//     PlcTask Inputs/GVL_iXlinker.EtherCAT_Master_ERxxxx.Beckhoff_ER6xxx.Beckhoff_ER6xxxEK1122.A_0005_ER6002_0002_0023.COM_TxPDO_Map_Inputs_Channel_2.Data_In[12] <-> COM TxPDO-Map Inputs Channel 2/Data In 12
//     PlcTask Inputs/GVL_iXlinker.EtherCAT_Master_ERxxxx.Beckhoff_ER6xxx.Beckhoff_ER6xxxEK1122.A_0005_ER6002_0002_0023.COM_TxPDO_Map_Inputs_Channel_2.Data_In[13] <-> COM TxPDO-Map Inputs Channel 2/Data In 13
//     PlcTask Inputs/GVL_iXlinker.EtherCAT_Master_ERxxxx.Beckhoff_ER6xxx.Beckhoff_ER6xxxEK1122.A_0005_ER6002_0002_0023.COM_TxPDO_Map_Inputs_Channel_2.Data_In[14] <-> COM TxPDO-Map Inputs Channel 2/Data In 14
//     PlcTask Inputs/GVL_iXlinker.EtherCAT_Master_ERxxxx.Beckhoff_ER6xxx.Beckhoff_ER6xxxEK1122.A_0005_ER6002_0002_0023.COM_TxPDO_Map_Inputs_Channel_2.Data_In[15] <-> COM TxPDO-Map Inputs Channel 2/Data In 15
//     PlcTask Inputs/GVL_iXlinker.EtherCAT_Master_ERxxxx.Beckhoff_ER6xxx.Beckhoff_ER6xxxEK1122.A_0005_ER6002_0002_0023.COM_TxPDO_Map_Inputs_Channel_2.Data_In[16] <-> COM TxPDO-Map Inputs Channel 2/Data In 16
//     PlcTask Inputs/GVL_iXlinker.EtherCAT_Master_ERxxxx.Beckhoff_ER6xxx.Beckhoff_ER6xxxEK1122.A_0005_ER6002_0002_0023.COM_TxPDO_Map_Inputs_Channel_2.Data_In[17] <-> COM TxPDO-Map Inputs Channel 2/Data In 17
//     PlcTask Inputs/GVL_iXlinker.EtherCAT_Master_ERxxxx.Beckhoff_ER6xxx.Beckhoff_ER6xxxEK1122.A_0005_ER6002_0002_0023.COM_TxPDO_Map_Inputs_Channel_2.Data_In[18] <-> COM TxPDO-Map Inputs Channel 2/Data In 18
//     PlcTask Inputs/GVL_iXlinker.EtherCAT_Master_ERxxxx.Beckhoff_ER6xxx.Beckhoff_ER6xxxEK1122.A_0005_ER6002_0002_0023.COM_TxPDO_Map_Inputs_Channel_2.Data_In[19] <-> COM TxPDO-Map Inputs Channel 2/Data In 19
//     PlcTask Inputs/GVL_iXlinker.EtherCAT_Master_ERxxxx.Beckhoff_ER6xxx.Beckhoff_ER6xxxEK1122.A_0005_ER6002_0002_0023.COM_TxPDO_Map_Inputs_Channel_2.Data_In[20] <-> COM TxPDO-Map Inputs Channel 2/Data In 20
//     PlcTask Inputs/GVL_iXlinker.EtherCAT_Master_ERxxxx.Beckhoff_ER6xxx.Beckhoff_ER6xxxEK1122.A_0005_ER6002_0002_0023.COM_TxPDO_Map_Inputs_Channel_2.Data_In[21] <-> COM TxPDO-Map Inputs Channel 2/Data In 21
//     PlcTask Outputs/GVL_iXlinker.EtherCAT_Master_ERxxxx.Beckhoff_ER6xxx.Beckhoff_ER6xxxEK1122.A_0005_ER6002_0002_0023.COM_RxPDO_Map_Outputs_Channel_1.Ctrl <-> COM RxPDO-Map Outputs Channel 1/Ctrl
//     PlcTask Outputs/GVL_iXlinker.EtherCAT_Master_ERxxxx.Beckhoff_ER6xxx.Beckhoff_ER6xxxEK1122.A_0005_ER6002_0002_0023.COM_RxPDO_Map_Outputs_Channel_2.Ctrl <-> COM RxPDO-Map Outputs Channel 2/Ctrl
//     PlcTask Outputs/GVL_iXlinker.EtherCAT_Master_ERxxxx.Beckhoff_ER6xxx.Beckhoff_ER6xxxEK1122.A_0005_ER6002_0002_0023.COM_RxPDO_Map_Outputs_Channel_1.Data_Out[0] <-> COM RxPDO-Map Outputs Channel 1/Data Out 0
//     PlcTask Outputs/GVL_iXlinker.EtherCAT_Master_ERxxxx.Beckhoff_ER6xxx.Beckhoff_ER6xxxEK1122.A_0005_ER6002_0002_0023.COM_RxPDO_Map_Outputs_Channel_1.Data_Out[1] <-> COM RxPDO-Map Outputs Channel 1/Data Out 1
//     PlcTask Outputs/GVL_iXlinker.EtherCAT_Master_ERxxxx.Beckhoff_ER6xxx.Beckhoff_ER6xxxEK1122.A_0005_ER6002_0002_0023.COM_RxPDO_Map_Outputs_Channel_1.Data_Out[2] <-> COM RxPDO-Map Outputs Channel 1/Data Out 2
//     PlcTask Outputs/GVL_iXlinker.EtherCAT_Master_ERxxxx.Beckhoff_ER6xxx.Beckhoff_ER6xxxEK1122.A_0005_ER6002_0002_0023.COM_RxPDO_Map_Outputs_Channel_1.Data_Out[3] <-> COM RxPDO-Map Outputs Channel 1/Data Out 3
//     PlcTask Outputs/GVL_iXlinker.EtherCAT_Master_ERxxxx.Beckhoff_ER6xxx.Beckhoff_ER6xxxEK1122.A_0005_ER6002_0002_0023.COM_RxPDO_Map_Outputs_Channel_1.Data_Out[4] <-> COM RxPDO-Map Outputs Channel 1/Data Out 4
//     PlcTask Outputs/GVL_iXlinker.EtherCAT_Master_ERxxxx.Beckhoff_ER6xxx.Beckhoff_ER6xxxEK1122.A_0005_ER6002_0002_0023.COM_RxPDO_Map_Outputs_Channel_1.Data_Out[5] <-> COM RxPDO-Map Outputs Channel 1/Data Out 5
//     PlcTask Outputs/GVL_iXlinker.EtherCAT_Master_ERxxxx.Beckhoff_ER6xxx.Beckhoff_ER6xxxEK1122.A_0005_ER6002_0002_0023.COM_RxPDO_Map_Outputs_Channel_1.Data_Out[6] <-> COM RxPDO-Map Outputs Channel 1/Data Out 6
//     PlcTask Outputs/GVL_iXlinker.EtherCAT_Master_ERxxxx.Beckhoff_ER6xxx.Beckhoff_ER6xxxEK1122.A_0005_ER6002_0002_0023.COM_RxPDO_Map_Outputs_Channel_1.Data_Out[7] <-> COM RxPDO-Map Outputs Channel 1/Data Out 7
//     PlcTask Outputs/GVL_iXlinker.EtherCAT_Master_ERxxxx.Beckhoff_ER6xxx.Beckhoff_ER6xxxEK1122.A_0005_ER6002_0002_0023.COM_RxPDO_Map_Outputs_Channel_1.Data_Out[8] <-> COM RxPDO-Map Outputs Channel 1/Data Out 8
//     PlcTask Outputs/GVL_iXlinker.EtherCAT_Master_ERxxxx.Beckhoff_ER6xxx.Beckhoff_ER6xxxEK1122.A_0005_ER6002_0002_0023.COM_RxPDO_Map_Outputs_Channel_1.Data_Out[9] <-> COM RxPDO-Map Outputs Channel 1/Data Out 9
//     PlcTask Outputs/GVL_iXlinker.EtherCAT_Master_ERxxxx.Beckhoff_ER6xxx.Beckhoff_ER6xxxEK1122.A_0005_ER6002_0002_0023.COM_RxPDO_Map_Outputs_Channel_1.Data_Out[10] <-> COM RxPDO-Map Outputs Channel 1/Data Out 10
//     PlcTask Outputs/GVL_iXlinker.EtherCAT_Master_ERxxxx.Beckhoff_ER6xxx.Beckhoff_ER6xxxEK1122.A_0005_ER6002_0002_0023.COM_RxPDO_Map_Outputs_Channel_1.Data_Out[11] <-> COM RxPDO-Map Outputs Channel 1/Data Out 11
//     PlcTask Outputs/GVL_iXlinker.EtherCAT_Master_ERxxxx.Beckhoff_ER6xxx.Beckhoff_ER6xxxEK1122.A_0005_ER6002_0002_0023.COM_RxPDO_Map_Outputs_Channel_1.Data_Out[12] <-> COM RxPDO-Map Outputs Channel 1/Data Out 12
//     PlcTask Outputs/GVL_iXlinker.EtherCAT_Master_ERxxxx.Beckhoff_ER6xxx.Beckhoff_ER6xxxEK1122.A_0005_ER6002_0002_0023.COM_RxPDO_Map_Outputs_Channel_1.Data_Out[13] <-> COM RxPDO-Map Outputs Channel 1/Data Out 13
//     PlcTask Outputs/GVL_iXlinker.EtherCAT_Master_ERxxxx.Beckhoff_ER6xxx.Beckhoff_ER6xxxEK1122.A_0005_ER6002_0002_0023.COM_RxPDO_Map_Outputs_Channel_1.Data_Out[14] <-> COM RxPDO-Map Outputs Channel 1/Data Out 14
//     PlcTask Outputs/GVL_iXlinker.EtherCAT_Master_ERxxxx.Beckhoff_ER6xxx.Beckhoff_ER6xxxEK1122.A_0005_ER6002_0002_0023.COM_RxPDO_Map_Outputs_Channel_1.Data_Out[15] <-> COM RxPDO-Map Outputs Channel 1/Data Out 15
//     PlcTask Outputs/GVL_iXlinker.EtherCAT_Master_ERxxxx.Beckhoff_ER6xxx.Beckhoff_ER6xxxEK1122.A_0005_ER6002_0002_0023.COM_RxPDO_Map_Outputs_Channel_1.Data_Out[16] <-> COM RxPDO-Map Outputs Channel 1/Data Out 16
//     PlcTask Outputs/GVL_iXlinker.EtherCAT_Master_ERxxxx.Beckhoff_ER6xxx.Beckhoff_ER6xxxEK1122.A_0005_ER6002_0002_0023.COM_RxPDO_Map_Outputs_Channel_1.Data_Out[17] <-> COM RxPDO-Map Outputs Channel 1/Data Out 17
//     PlcTask Outputs/GVL_iXlinker.EtherCAT_Master_ERxxxx.Beckhoff_ER6xxx.Beckhoff_ER6xxxEK1122.A_0005_ER6002_0002_0023.COM_RxPDO_Map_Outputs_Channel_1.Data_Out[18] <-> COM RxPDO-Map Outputs Channel 1/Data Out 18
//     PlcTask Outputs/GVL_iXlinker.EtherCAT_Master_ERxxxx.Beckhoff_ER6xxx.Beckhoff_ER6xxxEK1122.A_0005_ER6002_0002_0023.COM_RxPDO_Map_Outputs_Channel_1.Data_Out[19] <-> COM RxPDO-Map Outputs Channel 1/Data Out 19
//     PlcTask Outputs/GVL_iXlinker.EtherCAT_Master_ERxxxx.Beckhoff_ER6xxx.Beckhoff_ER6xxxEK1122.A_0005_ER6002_0002_0023.COM_RxPDO_Map_Outputs_Channel_1.Data_Out[20] <-> COM RxPDO-Map Outputs Channel 1/Data Out 20
//     PlcTask Outputs/GVL_iXlinker.EtherCAT_Master_ERxxxx.Beckhoff_ER6xxx.Beckhoff_ER6xxxEK1122.A_0005_ER6002_0002_0023.COM_RxPDO_Map_Outputs_Channel_1.Data_Out[21] <-> COM RxPDO-Map Outputs Channel 1/Data Out 21
//     PlcTask Outputs/GVL_iXlinker.EtherCAT_Master_ERxxxx.Beckhoff_ER6xxx.Beckhoff_ER6xxxEK1122.A_0005_ER6002_0002_0023.COM_RxPDO_Map_Outputs_Channel_2.Data_Out[0] <-> COM RxPDO-Map Outputs Channel 2/Data Out 0
//     PlcTask Outputs/GVL_iXlinker.EtherCAT_Master_ERxxxx.Beckhoff_ER6xxx.Beckhoff_ER6xxxEK1122.A_0005_ER6002_0002_0023.COM_RxPDO_Map_Outputs_Channel_2.Data_Out[1] <-> COM RxPDO-Map Outputs Channel 2/Data Out 1
//     PlcTask Outputs/GVL_iXlinker.EtherCAT_Master_ERxxxx.Beckhoff_ER6xxx.Beckhoff_ER6xxxEK1122.A_0005_ER6002_0002_0023.COM_RxPDO_Map_Outputs_Channel_2.Data_Out[2] <-> COM RxPDO-Map Outputs Channel 2/Data Out 2
//     PlcTask Outputs/GVL_iXlinker.EtherCAT_Master_ERxxxx.Beckhoff_ER6xxx.Beckhoff_ER6xxxEK1122.A_0005_ER6002_0002_0023.COM_RxPDO_Map_Outputs_Channel_2.Data_Out[3] <-> COM RxPDO-Map Outputs Channel 2/Data Out 3
//     PlcTask Outputs/GVL_iXlinker.EtherCAT_Master_ERxxxx.Beckhoff_ER6xxx.Beckhoff_ER6xxxEK1122.A_0005_ER6002_0002_0023.COM_RxPDO_Map_Outputs_Channel_2.Data_Out[4] <-> COM RxPDO-Map Outputs Channel 2/Data Out 4
//     PlcTask Outputs/GVL_iXlinker.EtherCAT_Master_ERxxxx.Beckhoff_ER6xxx.Beckhoff_ER6xxxEK1122.A_0005_ER6002_0002_0023.COM_RxPDO_Map_Outputs_Channel_2.Data_Out[5] <-> COM RxPDO-Map Outputs Channel 2/Data Out 5
//     PlcTask Outputs/GVL_iXlinker.EtherCAT_Master_ERxxxx.Beckhoff_ER6xxx.Beckhoff_ER6xxxEK1122.A_0005_ER6002_0002_0023.COM_RxPDO_Map_Outputs_Channel_2.Data_Out[6] <-> COM RxPDO-Map Outputs Channel 2/Data Out 6
//     PlcTask Outputs/GVL_iXlinker.EtherCAT_Master_ERxxxx.Beckhoff_ER6xxx.Beckhoff_ER6xxxEK1122.A_0005_ER6002_0002_0023.COM_RxPDO_Map_Outputs_Channel_2.Data_Out[7] <-> COM RxPDO-Map Outputs Channel 2/Data Out 7
//     PlcTask Outputs/GVL_iXlinker.EtherCAT_Master_ERxxxx.Beckhoff_ER6xxx.Beckhoff_ER6xxxEK1122.A_0005_ER6002_0002_0023.COM_RxPDO_Map_Outputs_Channel_2.Data_Out[8] <-> COM RxPDO-Map Outputs Channel 2/Data Out 8
//     PlcTask Outputs/GVL_iXlinker.EtherCAT_Master_ERxxxx.Beckhoff_ER6xxx.Beckhoff_ER6xxxEK1122.A_0005_ER6002_0002_0023.COM_RxPDO_Map_Outputs_Channel_2.Data_Out[9] <-> COM RxPDO-Map Outputs Channel 2/Data Out 9
//     PlcTask Outputs/GVL_iXlinker.EtherCAT_Master_ERxxxx.Beckhoff_ER6xxx.Beckhoff_ER6xxxEK1122.A_0005_ER6002_0002_0023.COM_RxPDO_Map_Outputs_Channel_2.Data_Out[10] <-> COM RxPDO-Map Outputs Channel 2/Data Out 10
//     PlcTask Outputs/GVL_iXlinker.EtherCAT_Master_ERxxxx.Beckhoff_ER6xxx.Beckhoff_ER6xxxEK1122.A_0005_ER6002_0002_0023.COM_RxPDO_Map_Outputs_Channel_2.Data_Out[11] <-> COM RxPDO-Map Outputs Channel 2/Data Out 11
//     PlcTask Outputs/GVL_iXlinker.EtherCAT_Master_ERxxxx.Beckhoff_ER6xxx.Beckhoff_ER6xxxEK1122.A_0005_ER6002_0002_0023.COM_RxPDO_Map_Outputs_Channel_2.Data_Out[12] <-> COM RxPDO-Map Outputs Channel 2/Data Out 12
//     PlcTask Outputs/GVL_iXlinker.EtherCAT_Master_ERxxxx.Beckhoff_ER6xxx.Beckhoff_ER6xxxEK1122.A_0005_ER6002_0002_0023.COM_RxPDO_Map_Outputs_Channel_2.Data_Out[13] <-> COM RxPDO-Map Outputs Channel 2/Data Out 13
//     PlcTask Outputs/GVL_iXlinker.EtherCAT_Master_ERxxxx.Beckhoff_ER6xxx.Beckhoff_ER6xxxEK1122.A_0005_ER6002_0002_0023.COM_RxPDO_Map_Outputs_Channel_2.Data_Out[14] <-> COM RxPDO-Map Outputs Channel 2/Data Out 14
//     PlcTask Outputs/GVL_iXlinker.EtherCAT_Master_ERxxxx.Beckhoff_ER6xxx.Beckhoff_ER6xxxEK1122.A_0005_ER6002_0002_0023.COM_RxPDO_Map_Outputs_Channel_2.Data_Out[15] <-> COM RxPDO-Map Outputs Channel 2/Data Out 15
//     PlcTask Outputs/GVL_iXlinker.EtherCAT_Master_ERxxxx.Beckhoff_ER6xxx.Beckhoff_ER6xxxEK1122.A_0005_ER6002_0002_0023.COM_RxPDO_Map_Outputs_Channel_2.Data_Out[16] <-> COM RxPDO-Map Outputs Channel 2/Data Out 16
//     PlcTask Outputs/GVL_iXlinker.EtherCAT_Master_ERxxxx.Beckhoff_ER6xxx.Beckhoff_ER6xxxEK1122.A_0005_ER6002_0002_0023.COM_RxPDO_Map_Outputs_Channel_2.Data_Out[17] <-> COM RxPDO-Map Outputs Channel 2/Data Out 17
//     PlcTask Outputs/GVL_iXlinker.EtherCAT_Master_ERxxxx.Beckhoff_ER6xxx.Beckhoff_ER6xxxEK1122.A_0005_ER6002_0002_0023.COM_RxPDO_Map_Outputs_Channel_2.Data_Out[18] <-> COM RxPDO-Map Outputs Channel 2/Data Out 18
//     PlcTask Outputs/GVL_iXlinker.EtherCAT_Master_ERxxxx.Beckhoff_ER6xxx.Beckhoff_ER6xxxEK1122.A_0005_ER6002_0002_0023.COM_RxPDO_Map_Outputs_Channel_2.Data_Out[19] <-> COM RxPDO-Map Outputs Channel 2/Data Out 19
//     PlcTask Outputs/GVL_iXlinker.EtherCAT_Master_ERxxxx.Beckhoff_ER6xxx.Beckhoff_ER6xxxEK1122.A_0005_ER6002_0002_0023.COM_RxPDO_Map_Outputs_Channel_2.Data_Out[20] <-> COM RxPDO-Map Outputs Channel 2/Data Out 20
//     PlcTask Outputs/GVL_iXlinker.EtherCAT_Master_ERxxxx.Beckhoff_ER6xxx.Beckhoff_ER6xxxEK1122.A_0005_ER6002_0002_0023.COM_RxPDO_Map_Outputs_Channel_2.Data_Out[21] <-> COM RxPDO-Map Outputs Channel 2/Data Out 21
//     PlcTask Inputs/GVL_iXlinker.EtherCAT_Master_ERxxxx.Beckhoff_ER6xxx.Beckhoff_ER6xxxEK1122.A_0005_ER6002_0002_0023.WcState.WcState <-> WcState/WcState
//     PlcTask Inputs/GVL_iXlinker.EtherCAT_Master_ERxxxx.Beckhoff_ER6xxx.Beckhoff_ER6xxxEK1122.A_0005_ER6002_0002_0023.WcState.InputToggle <-> WcState/InputToggle
//     PlcTask Inputs/GVL_iXlinker.EtherCAT_Master_ERxxxx.Beckhoff_ER6xxx.Beckhoff_ER6xxxEK1122.A_0005_ER6002_0002_0023.InfoData.AdsAddr <-> InfoData/AdsAddr
//     PlcTask Inputs/GVL_iXlinker.EtherCAT_Master_ERxxxx.Beckhoff_ER6xxx.Beckhoff_ER6xxxEK1122.A_0005_ER6002_0002_0023.InfoData.State <-> InfoData/State
//   PLC/PLC Instance <-> EtherCAT Master ERxxxx/Beckhoff ER7xxx
//     PlcTask Inputs/GVL_iXlinker.EtherCAT_Master_ERxxxx.Beckhoff_ER7xxx.InfoData.State <-> InfoData/State
//   PLC/PLC Instance <-> EtherCAT Master ERxxxx/Beckhoff ER7xxx/Beckhoff ER7xxxEK1122
//     PlcTask Inputs/GVL_iXlinker.EtherCAT_Master_ERxxxx.Beckhoff_ER7xxx.Beckhoff_ER7xxxEK1122.InfoData.State <-> InfoData/State
//   PLC/PLC Instance <-> EtherCAT Master ERxxxx/Beckhoff ER7xxx/Beckhoff ER7xxxEK1122/Beckhoff ER7xxxsub EK1100
//     PlcTask Inputs/GVL_iXlinker.EtherCAT_Master_ERxxxx.Beckhoff_ER7xxx.Beckhoff_ER7xxxEK1122.Beckhoff_ER7xxxsub_EK1100.InfoData.State <-> InfoData/State
//   PLC/PLC Instance <-> EtherCAT Master ERxxxx/Beckhoff ER7xxx/Beckhoff ER7xxxEK1122/A_0001(ER7041-0002-0024)
//     PlcTask Inputs/GVL_iXlinker.EtherCAT_Master_ERxxxx.Beckhoff_ER7xxx.Beckhoff_ER7xxxEK1122.A_0001_ER7041_0002_0024.ENC_Status_compact.Status/Latch_C_valid <-> ENC Status compact/Status/Latch C valid
//     PlcTask Inputs/GVL_iXlinker.EtherCAT_Master_ERxxxx.Beckhoff_ER7xxx.Beckhoff_ER7xxxEK1122.A_0001_ER7041_0002_0024.ENC_Status_compact.Status/Latch_extern_valid <-> ENC Status compact/Status/Latch extern valid
//     PlcTask Inputs/GVL_iXlinker.EtherCAT_Master_ERxxxx.Beckhoff_ER7xxx.Beckhoff_ER7xxxEK1122.A_0001_ER7041_0002_0024.ENC_Status_compact.Status/Set_counter_done <-> ENC Status compact/Status/Set counter done
//     PlcTask Inputs/GVL_iXlinker.EtherCAT_Master_ERxxxx.Beckhoff_ER7xxx.Beckhoff_ER7xxxEK1122.A_0001_ER7041_0002_0024.ENC_Status_compact.Status/Counter_underflow <-> ENC Status compact/Status/Counter underflow
//     PlcTask Inputs/GVL_iXlinker.EtherCAT_Master_ERxxxx.Beckhoff_ER7xxx.Beckhoff_ER7xxxEK1122.A_0001_ER7041_0002_0024.ENC_Status_compact.Status/Counter_overflow <-> ENC Status compact/Status/Counter overflow
//     PlcTask Inputs/GVL_iXlinker.EtherCAT_Master_ERxxxx.Beckhoff_ER7xxx.Beckhoff_ER7xxxEK1122.A_0001_ER7041_0002_0024.ENC_Status_compact.Status/Extrapolation_stall <-> ENC Status compact/Status/Extrapolation stall
//     PlcTask Inputs/GVL_iXlinker.EtherCAT_Master_ERxxxx.Beckhoff_ER7xxx.Beckhoff_ER7xxxEK1122.A_0001_ER7041_0002_0024.ENC_Status_compact.Status/Status_of_input_A <-> ENC Status compact/Status/Status of input A
//     PlcTask Inputs/GVL_iXlinker.EtherCAT_Master_ERxxxx.Beckhoff_ER7xxx.Beckhoff_ER7xxxEK1122.A_0001_ER7041_0002_0024.ENC_Status_compact.Status/Status_of_input_B <-> ENC Status compact/Status/Status of input B
//     PlcTask Inputs/GVL_iXlinker.EtherCAT_Master_ERxxxx.Beckhoff_ER7xxx.Beckhoff_ER7xxxEK1122.A_0001_ER7041_0002_0024.ENC_Status_compact.Status/Status_of_input_C <-> ENC Status compact/Status/Status of input C
//     PlcTask Inputs/GVL_iXlinker.EtherCAT_Master_ERxxxx.Beckhoff_ER7xxx.Beckhoff_ER7xxxEK1122.A_0001_ER7041_0002_0024.ENC_Status_compact.Status/Status_of_extern_latch <-> ENC Status compact/Status/Status of extern latch
//     PlcTask Inputs/GVL_iXlinker.EtherCAT_Master_ERxxxx.Beckhoff_ER7xxx.Beckhoff_ER7xxxEK1122.A_0001_ER7041_0002_0024.ENC_Status_compact.Status/Sync_error <-> ENC Status compact/Status/Sync error
//     PlcTask Inputs/GVL_iXlinker.EtherCAT_Master_ERxxxx.Beckhoff_ER7xxx.Beckhoff_ER7xxxEK1122.A_0001_ER7041_0002_0024.ENC_Status_compact.Status/TxPDO_Toggle <-> ENC Status compact/Status/TxPDO Toggle
//     PlcTask Inputs/GVL_iXlinker.EtherCAT_Master_ERxxxx.Beckhoff_ER7xxx.Beckhoff_ER7xxxEK1122.A_0001_ER7041_0002_0024.ENC_Status_compact.Counter_value <-> ENC Status compact/Counter value
//     PlcTask Inputs/GVL_iXlinker.EtherCAT_Master_ERxxxx.Beckhoff_ER7xxx.Beckhoff_ER7xxxEK1122.A_0001_ER7041_0002_0024.ENC_Status_compact.Latch_value <-> ENC Status compact/Latch value
//     PlcTask Inputs/GVL_iXlinker.EtherCAT_Master_ERxxxx.Beckhoff_ER7xxx.Beckhoff_ER7xxxEK1122.A_0001_ER7041_0002_0024.STM_Status.Status/Ready_to_enable <-> STM Status/Status/Ready to enable
//     PlcTask Inputs/GVL_iXlinker.EtherCAT_Master_ERxxxx.Beckhoff_ER7xxx.Beckhoff_ER7xxxEK1122.A_0001_ER7041_0002_0024.STM_Status.Status/Ready <-> STM Status/Status/Ready
//     PlcTask Inputs/GVL_iXlinker.EtherCAT_Master_ERxxxx.Beckhoff_ER7xxx.Beckhoff_ER7xxxEK1122.A_0001_ER7041_0002_0024.STM_Status.Status/Warning <-> STM Status/Status/Warning
//     PlcTask Inputs/GVL_iXlinker.EtherCAT_Master_ERxxxx.Beckhoff_ER7xxx.Beckhoff_ER7xxxEK1122.A_0001_ER7041_0002_0024.STM_Status.Status/Error <-> STM Status/Status/Error
//     PlcTask Inputs/GVL_iXlinker.EtherCAT_Master_ERxxxx.Beckhoff_ER7xxx.Beckhoff_ER7xxxEK1122.A_0001_ER7041_0002_0024.STM_Status.Status/Moving_positive <-> STM Status/Status/Moving positive
//     PlcTask Inputs/GVL_iXlinker.EtherCAT_Master_ERxxxx.Beckhoff_ER7xxx.Beckhoff_ER7xxxEK1122.A_0001_ER7041_0002_0024.STM_Status.Status/Moving_negative <-> STM Status/Status/Moving negative
//     PlcTask Inputs/GVL_iXlinker.EtherCAT_Master_ERxxxx.Beckhoff_ER7xxx.Beckhoff_ER7xxxEK1122.A_0001_ER7041_0002_0024.STM_Status.Status/Torque_reduced <-> STM Status/Status/Torque reduced
//     PlcTask Inputs/GVL_iXlinker.EtherCAT_Master_ERxxxx.Beckhoff_ER7xxx.Beckhoff_ER7xxxEK1122.A_0001_ER7041_0002_0024.STM_Status.Status/Digital_input_1 <-> STM Status/Status/Digital input 1
//     PlcTask Inputs/GVL_iXlinker.EtherCAT_Master_ERxxxx.Beckhoff_ER7xxx.Beckhoff_ER7xxxEK1122.A_0001_ER7041_0002_0024.STM_Status.Status/Digital_input_2 <-> STM Status/Status/Digital input 2
//     PlcTask Inputs/GVL_iXlinker.EtherCAT_Master_ERxxxx.Beckhoff_ER7xxx.Beckhoff_ER7xxxEK1122.A_0001_ER7041_0002_0024.STM_Status.Status/Sync_error <-> STM Status/Status/Sync error
//     PlcTask Inputs/GVL_iXlinker.EtherCAT_Master_ERxxxx.Beckhoff_ER7xxx.Beckhoff_ER7xxxEK1122.A_0001_ER7041_0002_0024.STM_Status.Status/TxPDO_Toggle <-> STM Status/Status/TxPDO Toggle
//     PlcTask Outputs/GVL_iXlinker.EtherCAT_Master_ERxxxx.Beckhoff_ER7xxx.Beckhoff_ER7xxxEK1122.A_0001_ER7041_0002_0024.ENC_Control_compact.Control/Enable_latch_C <-> ENC Control compact/Control/Enable latch C
//     PlcTask Outputs/GVL_iXlinker.EtherCAT_Master_ERxxxx.Beckhoff_ER7xxx.Beckhoff_ER7xxxEK1122.A_0001_ER7041_0002_0024.ENC_Control_compact.Control/Enable_latch_extern_on_positive_edge <-> ENC Control compact/Control/Enable latch extern on positive edge
//     PlcTask Outputs/GVL_iXlinker.EtherCAT_Master_ERxxxx.Beckhoff_ER7xxx.Beckhoff_ER7xxxEK1122.A_0001_ER7041_0002_0024.ENC_Control_compact.Control/Set_counter <-> ENC Control compact/Control/Set counter
//     PlcTask Outputs/GVL_iXlinker.EtherCAT_Master_ERxxxx.Beckhoff_ER7xxx.Beckhoff_ER7xxxEK1122.A_0001_ER7041_0002_0024.ENC_Control_compact.Control/Enable_latch_extern_on_negative_edge <-> ENC Control compact/Control/Enable latch extern on negative edge
//     PlcTask Outputs/GVL_iXlinker.EtherCAT_Master_ERxxxx.Beckhoff_ER7xxx.Beckhoff_ER7xxxEK1122.A_0001_ER7041_0002_0024.ENC_Control_compact.Set_counter_value <-> ENC Control compact/Set counter value
//     PlcTask Outputs/GVL_iXlinker.EtherCAT_Master_ERxxxx.Beckhoff_ER7xxx.Beckhoff_ER7xxxEK1122.A_0001_ER7041_0002_0024.STM_Control.Control/Enable <-> STM Control/Control/Enable
//     PlcTask Outputs/GVL_iXlinker.EtherCAT_Master_ERxxxx.Beckhoff_ER7xxx.Beckhoff_ER7xxxEK1122.A_0001_ER7041_0002_0024.STM_Control.Control/Reset <-> STM Control/Control/Reset
//     PlcTask Outputs/GVL_iXlinker.EtherCAT_Master_ERxxxx.Beckhoff_ER7xxx.Beckhoff_ER7xxxEK1122.A_0001_ER7041_0002_0024.STM_Control.Control/Reduce_torque <-> STM Control/Control/Reduce torque
//     PlcTask Outputs/GVL_iXlinker.EtherCAT_Master_ERxxxx.Beckhoff_ER7xxx.Beckhoff_ER7xxxEK1122.A_0001_ER7041_0002_0024.STM_Control.Control/Digital_output_1 <-> STM Control/Control/Digital output 1
//     PlcTask Outputs/GVL_iXlinker.EtherCAT_Master_ERxxxx.Beckhoff_ER7xxx.Beckhoff_ER7xxxEK1122.A_0001_ER7041_0002_0024.STM_Velocity.Velocity <-> STM Velocity/Velocity
//     PlcTask Inputs/GVL_iXlinker.EtherCAT_Master_ERxxxx.Beckhoff_ER7xxx.Beckhoff_ER7xxxEK1122.A_0001_ER7041_0002_0024.WcState.WcState <-> WcState/WcState
//     PlcTask Inputs/GVL_iXlinker.EtherCAT_Master_ERxxxx.Beckhoff_ER7xxx.Beckhoff_ER7xxxEK1122.A_0001_ER7041_0002_0024.WcState.InputToggle <-> WcState/InputToggle
//     PlcTask Inputs/GVL_iXlinker.EtherCAT_Master_ERxxxx.Beckhoff_ER7xxx.Beckhoff_ER7xxxEK1122.A_0001_ER7041_0002_0024.InfoData.AdsAddr <-> InfoData/AdsAddr
//     PlcTask Inputs/GVL_iXlinker.EtherCAT_Master_ERxxxx.Beckhoff_ER7xxx.Beckhoff_ER7xxxEK1122.A_0001_ER7041_0002_0024.InfoData.Chn0 <-> InfoData/Chn0
//     PlcTask Inputs/GVL_iXlinker.EtherCAT_Master_ERxxxx.Beckhoff_ER7xxx.Beckhoff_ER7xxxEK1122.A_0001_ER7041_0002_0024.InfoData.Chn1 <-> InfoData/Chn1
//     PlcTask Inputs/GVL_iXlinker.EtherCAT_Master_ERxxxx.Beckhoff_ER7xxx.Beckhoff_ER7xxxEK1122.A_0001_ER7041_0002_0024.InfoData.State <-> InfoData/State
//   PLC/PLC Instance <-> EtherCAT Master ERxxxx/Beckhoff ER7xxx/Beckhoff ER7xxxEK1122/A_0002(ER7041-0002-0025)
//     PlcTask Inputs/GVL_iXlinker.EtherCAT_Master_ERxxxx.Beckhoff_ER7xxx.Beckhoff_ER7xxxEK1122.A_0002_ER7041_0002_0025.ENC_Status_compact.Status/Latch_C_valid <-> ENC Status compact/Status/Latch C valid
//     PlcTask Inputs/GVL_iXlinker.EtherCAT_Master_ERxxxx.Beckhoff_ER7xxx.Beckhoff_ER7xxxEK1122.A_0002_ER7041_0002_0025.ENC_Status_compact.Status/Latch_extern_valid <-> ENC Status compact/Status/Latch extern valid
//     PlcTask Inputs/GVL_iXlinker.EtherCAT_Master_ERxxxx.Beckhoff_ER7xxx.Beckhoff_ER7xxxEK1122.A_0002_ER7041_0002_0025.ENC_Status_compact.Status/Set_counter_done <-> ENC Status compact/Status/Set counter done
//     PlcTask Inputs/GVL_iXlinker.EtherCAT_Master_ERxxxx.Beckhoff_ER7xxx.Beckhoff_ER7xxxEK1122.A_0002_ER7041_0002_0025.ENC_Status_compact.Status/Counter_underflow <-> ENC Status compact/Status/Counter underflow
//     PlcTask Inputs/GVL_iXlinker.EtherCAT_Master_ERxxxx.Beckhoff_ER7xxx.Beckhoff_ER7xxxEK1122.A_0002_ER7041_0002_0025.ENC_Status_compact.Status/Counter_overflow <-> ENC Status compact/Status/Counter overflow
//     PlcTask Inputs/GVL_iXlinker.EtherCAT_Master_ERxxxx.Beckhoff_ER7xxx.Beckhoff_ER7xxxEK1122.A_0002_ER7041_0002_0025.ENC_Status_compact.Status/Extrapolation_stall <-> ENC Status compact/Status/Extrapolation stall
//     PlcTask Inputs/GVL_iXlinker.EtherCAT_Master_ERxxxx.Beckhoff_ER7xxx.Beckhoff_ER7xxxEK1122.A_0002_ER7041_0002_0025.ENC_Status_compact.Status/Status_of_input_A <-> ENC Status compact/Status/Status of input A
//     PlcTask Inputs/GVL_iXlinker.EtherCAT_Master_ERxxxx.Beckhoff_ER7xxx.Beckhoff_ER7xxxEK1122.A_0002_ER7041_0002_0025.ENC_Status_compact.Status/Status_of_input_B <-> ENC Status compact/Status/Status of input B
//     PlcTask Inputs/GVL_iXlinker.EtherCAT_Master_ERxxxx.Beckhoff_ER7xxx.Beckhoff_ER7xxxEK1122.A_0002_ER7041_0002_0025.ENC_Status_compact.Status/Status_of_input_C <-> ENC Status compact/Status/Status of input C
//     PlcTask Inputs/GVL_iXlinker.EtherCAT_Master_ERxxxx.Beckhoff_ER7xxx.Beckhoff_ER7xxxEK1122.A_0002_ER7041_0002_0025.ENC_Status_compact.Status/Status_of_extern_latch <-> ENC Status compact/Status/Status of extern latch
//     PlcTask Inputs/GVL_iXlinker.EtherCAT_Master_ERxxxx.Beckhoff_ER7xxx.Beckhoff_ER7xxxEK1122.A_0002_ER7041_0002_0025.ENC_Status_compact.Status/Sync_error <-> ENC Status compact/Status/Sync error
//     PlcTask Inputs/GVL_iXlinker.EtherCAT_Master_ERxxxx.Beckhoff_ER7xxx.Beckhoff_ER7xxxEK1122.A_0002_ER7041_0002_0025.ENC_Status_compact.Status/TxPDO_Toggle <-> ENC Status compact/Status/TxPDO Toggle
//     PlcTask Inputs/GVL_iXlinker.EtherCAT_Master_ERxxxx.Beckhoff_ER7xxx.Beckhoff_ER7xxxEK1122.A_0002_ER7041_0002_0025.ENC_Status_compact.Counter_value <-> ENC Status compact/Counter value
//     PlcTask Inputs/GVL_iXlinker.EtherCAT_Master_ERxxxx.Beckhoff_ER7xxx.Beckhoff_ER7xxxEK1122.A_0002_ER7041_0002_0025.ENC_Status_compact.Latch_value <-> ENC Status compact/Latch value
//     PlcTask Inputs/GVL_iXlinker.EtherCAT_Master_ERxxxx.Beckhoff_ER7xxx.Beckhoff_ER7xxxEK1122.A_0002_ER7041_0002_0025.STM_Status.Status/Ready_to_enable <-> STM Status/Status/Ready to enable
//     PlcTask Inputs/GVL_iXlinker.EtherCAT_Master_ERxxxx.Beckhoff_ER7xxx.Beckhoff_ER7xxxEK1122.A_0002_ER7041_0002_0025.STM_Status.Status/Ready <-> STM Status/Status/Ready
//     PlcTask Inputs/GVL_iXlinker.EtherCAT_Master_ERxxxx.Beckhoff_ER7xxx.Beckhoff_ER7xxxEK1122.A_0002_ER7041_0002_0025.STM_Status.Status/Warning <-> STM Status/Status/Warning
//     PlcTask Inputs/GVL_iXlinker.EtherCAT_Master_ERxxxx.Beckhoff_ER7xxx.Beckhoff_ER7xxxEK1122.A_0002_ER7041_0002_0025.STM_Status.Status/Error <-> STM Status/Status/Error
//     PlcTask Inputs/GVL_iXlinker.EtherCAT_Master_ERxxxx.Beckhoff_ER7xxx.Beckhoff_ER7xxxEK1122.A_0002_ER7041_0002_0025.STM_Status.Status/Moving_positive <-> STM Status/Status/Moving positive
//     PlcTask Inputs/GVL_iXlinker.EtherCAT_Master_ERxxxx.Beckhoff_ER7xxx.Beckhoff_ER7xxxEK1122.A_0002_ER7041_0002_0025.STM_Status.Status/Moving_negative <-> STM Status/Status/Moving negative
//     PlcTask Inputs/GVL_iXlinker.EtherCAT_Master_ERxxxx.Beckhoff_ER7xxx.Beckhoff_ER7xxxEK1122.A_0002_ER7041_0002_0025.STM_Status.Status/Torque_reduced <-> STM Status/Status/Torque reduced
//     PlcTask Inputs/GVL_iXlinker.EtherCAT_Master_ERxxxx.Beckhoff_ER7xxx.Beckhoff_ER7xxxEK1122.A_0002_ER7041_0002_0025.STM_Status.Status/Digital_input_1 <-> STM Status/Status/Digital input 1
//     PlcTask Inputs/GVL_iXlinker.EtherCAT_Master_ERxxxx.Beckhoff_ER7xxx.Beckhoff_ER7xxxEK1122.A_0002_ER7041_0002_0025.STM_Status.Status/Digital_input_2 <-> STM Status/Status/Digital input 2
//     PlcTask Inputs/GVL_iXlinker.EtherCAT_Master_ERxxxx.Beckhoff_ER7xxx.Beckhoff_ER7xxxEK1122.A_0002_ER7041_0002_0025.STM_Status.Status/Sync_error <-> STM Status/Status/Sync error
//     PlcTask Inputs/GVL_iXlinker.EtherCAT_Master_ERxxxx.Beckhoff_ER7xxx.Beckhoff_ER7xxxEK1122.A_0002_ER7041_0002_0025.STM_Status.Status/TxPDO_Toggle <-> STM Status/Status/TxPDO Toggle
//     PlcTask Outputs/GVL_iXlinker.EtherCAT_Master_ERxxxx.Beckhoff_ER7xxx.Beckhoff_ER7xxxEK1122.A_0002_ER7041_0002_0025.ENC_Control_compact.Control/Enable_latch_C <-> ENC Control compact/Control/Enable latch C
//     PlcTask Outputs/GVL_iXlinker.EtherCAT_Master_ERxxxx.Beckhoff_ER7xxx.Beckhoff_ER7xxxEK1122.A_0002_ER7041_0002_0025.ENC_Control_compact.Control/Enable_latch_extern_on_positive_edge <-> ENC Control compact/Control/Enable latch extern on positive edge
//     PlcTask Outputs/GVL_iXlinker.EtherCAT_Master_ERxxxx.Beckhoff_ER7xxx.Beckhoff_ER7xxxEK1122.A_0002_ER7041_0002_0025.ENC_Control_compact.Control/Set_counter <-> ENC Control compact/Control/Set counter
//     PlcTask Outputs/GVL_iXlinker.EtherCAT_Master_ERxxxx.Beckhoff_ER7xxx.Beckhoff_ER7xxxEK1122.A_0002_ER7041_0002_0025.ENC_Control_compact.Control/Enable_latch_extern_on_negative_edge <-> ENC Control compact/Control/Enable latch extern on negative edge
//     PlcTask Outputs/GVL_iXlinker.EtherCAT_Master_ERxxxx.Beckhoff_ER7xxx.Beckhoff_ER7xxxEK1122.A_0002_ER7041_0002_0025.ENC_Control_compact.Set_counter_value <-> ENC Control compact/Set counter value
//     PlcTask Outputs/GVL_iXlinker.EtherCAT_Master_ERxxxx.Beckhoff_ER7xxx.Beckhoff_ER7xxxEK1122.A_0002_ER7041_0002_0025.STM_Control.Control/Enable <-> STM Control/Control/Enable
//     PlcTask Outputs/GVL_iXlinker.EtherCAT_Master_ERxxxx.Beckhoff_ER7xxx.Beckhoff_ER7xxxEK1122.A_0002_ER7041_0002_0025.STM_Control.Control/Reset <-> STM Control/Control/Reset
//     PlcTask Outputs/GVL_iXlinker.EtherCAT_Master_ERxxxx.Beckhoff_ER7xxx.Beckhoff_ER7xxxEK1122.A_0002_ER7041_0002_0025.STM_Control.Control/Reduce_torque <-> STM Control/Control/Reduce torque
//     PlcTask Outputs/GVL_iXlinker.EtherCAT_Master_ERxxxx.Beckhoff_ER7xxx.Beckhoff_ER7xxxEK1122.A_0002_ER7041_0002_0025.STM_Control.Control/Digital_output_1 <-> STM Control/Control/Digital output 1
//     PlcTask Outputs/GVL_iXlinker.EtherCAT_Master_ERxxxx.Beckhoff_ER7xxx.Beckhoff_ER7xxxEK1122.A_0002_ER7041_0002_0025.STM_Velocity.Velocity <-> STM Velocity/Velocity
//     PlcTask Inputs/GVL_iXlinker.EtherCAT_Master_ERxxxx.Beckhoff_ER7xxx.Beckhoff_ER7xxxEK1122.A_0002_ER7041_0002_0025.WcState.WcState <-> WcState/WcState
//     PlcTask Inputs/GVL_iXlinker.EtherCAT_Master_ERxxxx.Beckhoff_ER7xxx.Beckhoff_ER7xxxEK1122.A_0002_ER7041_0002_0025.WcState.InputToggle <-> WcState/InputToggle
//     PlcTask Inputs/GVL_iXlinker.EtherCAT_Master_ERxxxx.Beckhoff_ER7xxx.Beckhoff_ER7xxxEK1122.A_0002_ER7041_0002_0025.InfoData.AdsAddr <-> InfoData/AdsAddr
//     PlcTask Inputs/GVL_iXlinker.EtherCAT_Master_ERxxxx.Beckhoff_ER7xxx.Beckhoff_ER7xxxEK1122.A_0002_ER7041_0002_0025.InfoData.Chn0 <-> InfoData/Chn0
//     PlcTask Inputs/GVL_iXlinker.EtherCAT_Master_ERxxxx.Beckhoff_ER7xxx.Beckhoff_ER7xxxEK1122.A_0002_ER7041_0002_0025.InfoData.Chn1 <-> InfoData/Chn1
//     PlcTask Inputs/GVL_iXlinker.EtherCAT_Master_ERxxxx.Beckhoff_ER7xxx.Beckhoff_ER7xxxEK1122.A_0002_ER7041_0002_0025.InfoData.State <-> InfoData/State
//   PLC/PLC Instance <-> EtherCAT Master ERxxxx/Beckhoff ER7xxx/Beckhoff ER7xxxEK1122/A_0003(ER7041-1002-0024)
//     PlcTask Inputs/GVL_iXlinker.EtherCAT_Master_ERxxxx.Beckhoff_ER7xxx.Beckhoff_ER7xxxEK1122.A_0003_ER7041_1002_0024.ENC_Status_compact.Status/Latch_C_valid <-> ENC Status compact/Status/Latch C valid
//     PlcTask Inputs/GVL_iXlinker.EtherCAT_Master_ERxxxx.Beckhoff_ER7xxx.Beckhoff_ER7xxxEK1122.A_0003_ER7041_1002_0024.ENC_Status_compact.Status/Latch_extern_valid <-> ENC Status compact/Status/Latch extern valid
//     PlcTask Inputs/GVL_iXlinker.EtherCAT_Master_ERxxxx.Beckhoff_ER7xxx.Beckhoff_ER7xxxEK1122.A_0003_ER7041_1002_0024.ENC_Status_compact.Status/Set_counter_done <-> ENC Status compact/Status/Set counter done
//     PlcTask Inputs/GVL_iXlinker.EtherCAT_Master_ERxxxx.Beckhoff_ER7xxx.Beckhoff_ER7xxxEK1122.A_0003_ER7041_1002_0024.ENC_Status_compact.Status/Counter_underflow <-> ENC Status compact/Status/Counter underflow
//     PlcTask Inputs/GVL_iXlinker.EtherCAT_Master_ERxxxx.Beckhoff_ER7xxx.Beckhoff_ER7xxxEK1122.A_0003_ER7041_1002_0024.ENC_Status_compact.Status/Counter_overflow <-> ENC Status compact/Status/Counter overflow
//     PlcTask Inputs/GVL_iXlinker.EtherCAT_Master_ERxxxx.Beckhoff_ER7xxx.Beckhoff_ER7xxxEK1122.A_0003_ER7041_1002_0024.ENC_Status_compact.Status/Extrapolation_stall <-> ENC Status compact/Status/Extrapolation stall
//     PlcTask Inputs/GVL_iXlinker.EtherCAT_Master_ERxxxx.Beckhoff_ER7xxx.Beckhoff_ER7xxxEK1122.A_0003_ER7041_1002_0024.ENC_Status_compact.Status/Status_of_input_A <-> ENC Status compact/Status/Status of input A
//     PlcTask Inputs/GVL_iXlinker.EtherCAT_Master_ERxxxx.Beckhoff_ER7xxx.Beckhoff_ER7xxxEK1122.A_0003_ER7041_1002_0024.ENC_Status_compact.Status/Status_of_input_B <-> ENC Status compact/Status/Status of input B
//     PlcTask Inputs/GVL_iXlinker.EtherCAT_Master_ERxxxx.Beckhoff_ER7xxx.Beckhoff_ER7xxxEK1122.A_0003_ER7041_1002_0024.ENC_Status_compact.Status/Status_of_input_C <-> ENC Status compact/Status/Status of input C
//     PlcTask Inputs/GVL_iXlinker.EtherCAT_Master_ERxxxx.Beckhoff_ER7xxx.Beckhoff_ER7xxxEK1122.A_0003_ER7041_1002_0024.ENC_Status_compact.Status/Status_of_extern_latch <-> ENC Status compact/Status/Status of extern latch
//     PlcTask Inputs/GVL_iXlinker.EtherCAT_Master_ERxxxx.Beckhoff_ER7xxx.Beckhoff_ER7xxxEK1122.A_0003_ER7041_1002_0024.ENC_Status_compact.Status/Sync_error <-> ENC Status compact/Status/Sync error
//     PlcTask Inputs/GVL_iXlinker.EtherCAT_Master_ERxxxx.Beckhoff_ER7xxx.Beckhoff_ER7xxxEK1122.A_0003_ER7041_1002_0024.ENC_Status_compact.Status/TxPDO_Toggle <-> ENC Status compact/Status/TxPDO Toggle
//     PlcTask Inputs/GVL_iXlinker.EtherCAT_Master_ERxxxx.Beckhoff_ER7xxx.Beckhoff_ER7xxxEK1122.A_0003_ER7041_1002_0024.ENC_Status_compact.Counter_value <-> ENC Status compact/Counter value
//     PlcTask Inputs/GVL_iXlinker.EtherCAT_Master_ERxxxx.Beckhoff_ER7xxx.Beckhoff_ER7xxxEK1122.A_0003_ER7041_1002_0024.ENC_Status_compact.Latch_value <-> ENC Status compact/Latch value
//     PlcTask Inputs/GVL_iXlinker.EtherCAT_Master_ERxxxx.Beckhoff_ER7xxx.Beckhoff_ER7xxxEK1122.A_0003_ER7041_1002_0024.STM_Status.Status/Ready_to_enable <-> STM Status/Status/Ready to enable
//     PlcTask Inputs/GVL_iXlinker.EtherCAT_Master_ERxxxx.Beckhoff_ER7xxx.Beckhoff_ER7xxxEK1122.A_0003_ER7041_1002_0024.STM_Status.Status/Ready <-> STM Status/Status/Ready
//     PlcTask Inputs/GVL_iXlinker.EtherCAT_Master_ERxxxx.Beckhoff_ER7xxx.Beckhoff_ER7xxxEK1122.A_0003_ER7041_1002_0024.STM_Status.Status/Warning <-> STM Status/Status/Warning
//     PlcTask Inputs/GVL_iXlinker.EtherCAT_Master_ERxxxx.Beckhoff_ER7xxx.Beckhoff_ER7xxxEK1122.A_0003_ER7041_1002_0024.STM_Status.Status/Error <-> STM Status/Status/Error
//     PlcTask Inputs/GVL_iXlinker.EtherCAT_Master_ERxxxx.Beckhoff_ER7xxx.Beckhoff_ER7xxxEK1122.A_0003_ER7041_1002_0024.STM_Status.Status/Moving_positive <-> STM Status/Status/Moving positive
//     PlcTask Inputs/GVL_iXlinker.EtherCAT_Master_ERxxxx.Beckhoff_ER7xxx.Beckhoff_ER7xxxEK1122.A_0003_ER7041_1002_0024.STM_Status.Status/Moving_negative <-> STM Status/Status/Moving negative
//     PlcTask Inputs/GVL_iXlinker.EtherCAT_Master_ERxxxx.Beckhoff_ER7xxx.Beckhoff_ER7xxxEK1122.A_0003_ER7041_1002_0024.STM_Status.Status/Torque_reduced <-> STM Status/Status/Torque reduced
//     PlcTask Inputs/GVL_iXlinker.EtherCAT_Master_ERxxxx.Beckhoff_ER7xxx.Beckhoff_ER7xxxEK1122.A_0003_ER7041_1002_0024.STM_Status.Status/Digital_input_1 <-> STM Status/Status/Digital input 1
//     PlcTask Inputs/GVL_iXlinker.EtherCAT_Master_ERxxxx.Beckhoff_ER7xxx.Beckhoff_ER7xxxEK1122.A_0003_ER7041_1002_0024.STM_Status.Status/Digital_input_2 <-> STM Status/Status/Digital input 2
//     PlcTask Inputs/GVL_iXlinker.EtherCAT_Master_ERxxxx.Beckhoff_ER7xxx.Beckhoff_ER7xxxEK1122.A_0003_ER7041_1002_0024.STM_Status.Status/Sync_error <-> STM Status/Status/Sync error
//     PlcTask Inputs/GVL_iXlinker.EtherCAT_Master_ERxxxx.Beckhoff_ER7xxx.Beckhoff_ER7xxxEK1122.A_0003_ER7041_1002_0024.STM_Status.Status/TxPDO_Toggle <-> STM Status/Status/TxPDO Toggle
//     PlcTask Outputs/GVL_iXlinker.EtherCAT_Master_ERxxxx.Beckhoff_ER7xxx.Beckhoff_ER7xxxEK1122.A_0003_ER7041_1002_0024.ENC_Control_compact.Control/Enable_latch_C <-> ENC Control compact/Control/Enable latch C
//     PlcTask Outputs/GVL_iXlinker.EtherCAT_Master_ERxxxx.Beckhoff_ER7xxx.Beckhoff_ER7xxxEK1122.A_0003_ER7041_1002_0024.ENC_Control_compact.Control/Enable_latch_extern_on_positive_edge <-> ENC Control compact/Control/Enable latch extern on positive edge
//     PlcTask Outputs/GVL_iXlinker.EtherCAT_Master_ERxxxx.Beckhoff_ER7xxx.Beckhoff_ER7xxxEK1122.A_0003_ER7041_1002_0024.ENC_Control_compact.Control/Set_counter <-> ENC Control compact/Control/Set counter
//     PlcTask Outputs/GVL_iXlinker.EtherCAT_Master_ERxxxx.Beckhoff_ER7xxx.Beckhoff_ER7xxxEK1122.A_0003_ER7041_1002_0024.ENC_Control_compact.Control/Enable_latch_extern_on_negative_edge <-> ENC Control compact/Control/Enable latch extern on negative edge
//     PlcTask Outputs/GVL_iXlinker.EtherCAT_Master_ERxxxx.Beckhoff_ER7xxx.Beckhoff_ER7xxxEK1122.A_0003_ER7041_1002_0024.ENC_Control_compact.Set_counter_value <-> ENC Control compact/Set counter value
//     PlcTask Outputs/GVL_iXlinker.EtherCAT_Master_ERxxxx.Beckhoff_ER7xxx.Beckhoff_ER7xxxEK1122.A_0003_ER7041_1002_0024.STM_Control.Control/Enable <-> STM Control/Control/Enable
//     PlcTask Outputs/GVL_iXlinker.EtherCAT_Master_ERxxxx.Beckhoff_ER7xxx.Beckhoff_ER7xxxEK1122.A_0003_ER7041_1002_0024.STM_Control.Control/Reset <-> STM Control/Control/Reset
//     PlcTask Outputs/GVL_iXlinker.EtherCAT_Master_ERxxxx.Beckhoff_ER7xxx.Beckhoff_ER7xxxEK1122.A_0003_ER7041_1002_0024.STM_Control.Control/Reduce_torque <-> STM Control/Control/Reduce torque
//     PlcTask Outputs/GVL_iXlinker.EtherCAT_Master_ERxxxx.Beckhoff_ER7xxx.Beckhoff_ER7xxxEK1122.A_0003_ER7041_1002_0024.STM_Control.Control/Digital_output_1 <-> STM Control/Control/Digital output 1
//     PlcTask Outputs/GVL_iXlinker.EtherCAT_Master_ERxxxx.Beckhoff_ER7xxx.Beckhoff_ER7xxxEK1122.A_0003_ER7041_1002_0024.STM_Velocity.Velocity <-> STM Velocity/Velocity
//     PlcTask Inputs/GVL_iXlinker.EtherCAT_Master_ERxxxx.Beckhoff_ER7xxx.Beckhoff_ER7xxxEK1122.A_0003_ER7041_1002_0024.WcState.WcState <-> WcState/WcState
//     PlcTask Inputs/GVL_iXlinker.EtherCAT_Master_ERxxxx.Beckhoff_ER7xxx.Beckhoff_ER7xxxEK1122.A_0003_ER7041_1002_0024.WcState.InputToggle <-> WcState/InputToggle
//     PlcTask Inputs/GVL_iXlinker.EtherCAT_Master_ERxxxx.Beckhoff_ER7xxx.Beckhoff_ER7xxxEK1122.A_0003_ER7041_1002_0024.InfoData.AdsAddr <-> InfoData/AdsAddr
//     PlcTask Inputs/GVL_iXlinker.EtherCAT_Master_ERxxxx.Beckhoff_ER7xxx.Beckhoff_ER7xxxEK1122.A_0003_ER7041_1002_0024.InfoData.Chn0 <-> InfoData/Chn0
//     PlcTask Inputs/GVL_iXlinker.EtherCAT_Master_ERxxxx.Beckhoff_ER7xxx.Beckhoff_ER7xxxEK1122.A_0003_ER7041_1002_0024.InfoData.Chn1 <-> InfoData/Chn1
//     PlcTask Inputs/GVL_iXlinker.EtherCAT_Master_ERxxxx.Beckhoff_ER7xxx.Beckhoff_ER7xxxEK1122.A_0003_ER7041_1002_0024.InfoData.State <-> InfoData/State
//   PLC/PLC Instance <-> EtherCAT Master ERxxxx/Beckhoff ER7xxx/Beckhoff ER7xxxEK1122/A_0004(ER7041-1002-0025)
//     PlcTask Inputs/GVL_iXlinker.EtherCAT_Master_ERxxxx.Beckhoff_ER7xxx.Beckhoff_ER7xxxEK1122.A_0004_ER7041_1002_0025.ENC_Status_compact.Status/Latch_C_valid <-> ENC Status compact/Status/Latch C valid
//     PlcTask Inputs/GVL_iXlinker.EtherCAT_Master_ERxxxx.Beckhoff_ER7xxx.Beckhoff_ER7xxxEK1122.A_0004_ER7041_1002_0025.ENC_Status_compact.Status/Latch_extern_valid <-> ENC Status compact/Status/Latch extern valid
//     PlcTask Inputs/GVL_iXlinker.EtherCAT_Master_ERxxxx.Beckhoff_ER7xxx.Beckhoff_ER7xxxEK1122.A_0004_ER7041_1002_0025.ENC_Status_compact.Status/Set_counter_done <-> ENC Status compact/Status/Set counter done
//     PlcTask Inputs/GVL_iXlinker.EtherCAT_Master_ERxxxx.Beckhoff_ER7xxx.Beckhoff_ER7xxxEK1122.A_0004_ER7041_1002_0025.ENC_Status_compact.Status/Counter_underflow <-> ENC Status compact/Status/Counter underflow
//     PlcTask Inputs/GVL_iXlinker.EtherCAT_Master_ERxxxx.Beckhoff_ER7xxx.Beckhoff_ER7xxxEK1122.A_0004_ER7041_1002_0025.ENC_Status_compact.Status/Counter_overflow <-> ENC Status compact/Status/Counter overflow
//     PlcTask Inputs/GVL_iXlinker.EtherCAT_Master_ERxxxx.Beckhoff_ER7xxx.Beckhoff_ER7xxxEK1122.A_0004_ER7041_1002_0025.ENC_Status_compact.Status/Extrapolation_stall <-> ENC Status compact/Status/Extrapolation stall
//     PlcTask Inputs/GVL_iXlinker.EtherCAT_Master_ERxxxx.Beckhoff_ER7xxx.Beckhoff_ER7xxxEK1122.A_0004_ER7041_1002_0025.ENC_Status_compact.Status/Status_of_input_A <-> ENC Status compact/Status/Status of input A
//     PlcTask Inputs/GVL_iXlinker.EtherCAT_Master_ERxxxx.Beckhoff_ER7xxx.Beckhoff_ER7xxxEK1122.A_0004_ER7041_1002_0025.ENC_Status_compact.Status/Status_of_input_B <-> ENC Status compact/Status/Status of input B
//     PlcTask Inputs/GVL_iXlinker.EtherCAT_Master_ERxxxx.Beckhoff_ER7xxx.Beckhoff_ER7xxxEK1122.A_0004_ER7041_1002_0025.ENC_Status_compact.Status/Status_of_input_C <-> ENC Status compact/Status/Status of input C
//     PlcTask Inputs/GVL_iXlinker.EtherCAT_Master_ERxxxx.Beckhoff_ER7xxx.Beckhoff_ER7xxxEK1122.A_0004_ER7041_1002_0025.ENC_Status_compact.Status/Status_of_extern_latch <-> ENC Status compact/Status/Status of extern latch
//     PlcTask Inputs/GVL_iXlinker.EtherCAT_Master_ERxxxx.Beckhoff_ER7xxx.Beckhoff_ER7xxxEK1122.A_0004_ER7041_1002_0025.ENC_Status_compact.Status/Sync_error <-> ENC Status compact/Status/Sync error
//     PlcTask Inputs/GVL_iXlinker.EtherCAT_Master_ERxxxx.Beckhoff_ER7xxx.Beckhoff_ER7xxxEK1122.A_0004_ER7041_1002_0025.ENC_Status_compact.Status/TxPDO_Toggle <-> ENC Status compact/Status/TxPDO Toggle
//     PlcTask Inputs/GVL_iXlinker.EtherCAT_Master_ERxxxx.Beckhoff_ER7xxx.Beckhoff_ER7xxxEK1122.A_0004_ER7041_1002_0025.ENC_Status_compact.Counter_value <-> ENC Status compact/Counter value
//     PlcTask Inputs/GVL_iXlinker.EtherCAT_Master_ERxxxx.Beckhoff_ER7xxx.Beckhoff_ER7xxxEK1122.A_0004_ER7041_1002_0025.ENC_Status_compact.Latch_value <-> ENC Status compact/Latch value
//     PlcTask Inputs/GVL_iXlinker.EtherCAT_Master_ERxxxx.Beckhoff_ER7xxx.Beckhoff_ER7xxxEK1122.A_0004_ER7041_1002_0025.STM_Status.Status/Ready_to_enable <-> STM Status/Status/Ready to enable
//     PlcTask Inputs/GVL_iXlinker.EtherCAT_Master_ERxxxx.Beckhoff_ER7xxx.Beckhoff_ER7xxxEK1122.A_0004_ER7041_1002_0025.STM_Status.Status/Ready <-> STM Status/Status/Ready
//     PlcTask Inputs/GVL_iXlinker.EtherCAT_Master_ERxxxx.Beckhoff_ER7xxx.Beckhoff_ER7xxxEK1122.A_0004_ER7041_1002_0025.STM_Status.Status/Warning <-> STM Status/Status/Warning
//     PlcTask Inputs/GVL_iXlinker.EtherCAT_Master_ERxxxx.Beckhoff_ER7xxx.Beckhoff_ER7xxxEK1122.A_0004_ER7041_1002_0025.STM_Status.Status/Error <-> STM Status/Status/Error
//     PlcTask Inputs/GVL_iXlinker.EtherCAT_Master_ERxxxx.Beckhoff_ER7xxx.Beckhoff_ER7xxxEK1122.A_0004_ER7041_1002_0025.STM_Status.Status/Moving_positive <-> STM Status/Status/Moving positive
//     PlcTask Inputs/GVL_iXlinker.EtherCAT_Master_ERxxxx.Beckhoff_ER7xxx.Beckhoff_ER7xxxEK1122.A_0004_ER7041_1002_0025.STM_Status.Status/Moving_negative <-> STM Status/Status/Moving negative
//     PlcTask Inputs/GVL_iXlinker.EtherCAT_Master_ERxxxx.Beckhoff_ER7xxx.Beckhoff_ER7xxxEK1122.A_0004_ER7041_1002_0025.STM_Status.Status/Torque_reduced <-> STM Status/Status/Torque reduced
//     PlcTask Inputs/GVL_iXlinker.EtherCAT_Master_ERxxxx.Beckhoff_ER7xxx.Beckhoff_ER7xxxEK1122.A_0004_ER7041_1002_0025.STM_Status.Status/Digital_input_1 <-> STM Status/Status/Digital input 1
//     PlcTask Inputs/GVL_iXlinker.EtherCAT_Master_ERxxxx.Beckhoff_ER7xxx.Beckhoff_ER7xxxEK1122.A_0004_ER7041_1002_0025.STM_Status.Status/Digital_input_2 <-> STM Status/Status/Digital input 2
//     PlcTask Inputs/GVL_iXlinker.EtherCAT_Master_ERxxxx.Beckhoff_ER7xxx.Beckhoff_ER7xxxEK1122.A_0004_ER7041_1002_0025.STM_Status.Status/Sync_error <-> STM Status/Status/Sync error
//     PlcTask Inputs/GVL_iXlinker.EtherCAT_Master_ERxxxx.Beckhoff_ER7xxx.Beckhoff_ER7xxxEK1122.A_0004_ER7041_1002_0025.STM_Status.Status/TxPDO_Toggle <-> STM Status/Status/TxPDO Toggle
//     PlcTask Outputs/GVL_iXlinker.EtherCAT_Master_ERxxxx.Beckhoff_ER7xxx.Beckhoff_ER7xxxEK1122.A_0004_ER7041_1002_0025.ENC_Control_compact.Control/Enable_latch_C <-> ENC Control compact/Control/Enable latch C
//     PlcTask Outputs/GVL_iXlinker.EtherCAT_Master_ERxxxx.Beckhoff_ER7xxx.Beckhoff_ER7xxxEK1122.A_0004_ER7041_1002_0025.ENC_Control_compact.Control/Enable_latch_extern_on_positive_edge <-> ENC Control compact/Control/Enable latch extern on positive edge
//     PlcTask Outputs/GVL_iXlinker.EtherCAT_Master_ERxxxx.Beckhoff_ER7xxx.Beckhoff_ER7xxxEK1122.A_0004_ER7041_1002_0025.ENC_Control_compact.Control/Set_counter <-> ENC Control compact/Control/Set counter
//     PlcTask Outputs/GVL_iXlinker.EtherCAT_Master_ERxxxx.Beckhoff_ER7xxx.Beckhoff_ER7xxxEK1122.A_0004_ER7041_1002_0025.ENC_Control_compact.Control/Enable_latch_extern_on_negative_edge <-> ENC Control compact/Control/Enable latch extern on negative edge
//     PlcTask Outputs/GVL_iXlinker.EtherCAT_Master_ERxxxx.Beckhoff_ER7xxx.Beckhoff_ER7xxxEK1122.A_0004_ER7041_1002_0025.ENC_Control_compact.Set_counter_value <-> ENC Control compact/Set counter value
//     PlcTask Outputs/GVL_iXlinker.EtherCAT_Master_ERxxxx.Beckhoff_ER7xxx.Beckhoff_ER7xxxEK1122.A_0004_ER7041_1002_0025.STM_Control.Control/Enable <-> STM Control/Control/Enable
//     PlcTask Outputs/GVL_iXlinker.EtherCAT_Master_ERxxxx.Beckhoff_ER7xxx.Beckhoff_ER7xxxEK1122.A_0004_ER7041_1002_0025.STM_Control.Control/Reset <-> STM Control/Control/Reset
//     PlcTask Outputs/GVL_iXlinker.EtherCAT_Master_ERxxxx.Beckhoff_ER7xxx.Beckhoff_ER7xxxEK1122.A_0004_ER7041_1002_0025.STM_Control.Control/Reduce_torque <-> STM Control/Control/Reduce torque
//     PlcTask Outputs/GVL_iXlinker.EtherCAT_Master_ERxxxx.Beckhoff_ER7xxx.Beckhoff_ER7xxxEK1122.A_0004_ER7041_1002_0025.STM_Control.Control/Digital_output_1 <-> STM Control/Control/Digital output 1
//     PlcTask Outputs/GVL_iXlinker.EtherCAT_Master_ERxxxx.Beckhoff_ER7xxx.Beckhoff_ER7xxxEK1122.A_0004_ER7041_1002_0025.STM_Velocity.Velocity <-> STM Velocity/Velocity
//     PlcTask Inputs/GVL_iXlinker.EtherCAT_Master_ERxxxx.Beckhoff_ER7xxx.Beckhoff_ER7xxxEK1122.A_0004_ER7041_1002_0025.WcState.WcState <-> WcState/WcState
//     PlcTask Inputs/GVL_iXlinker.EtherCAT_Master_ERxxxx.Beckhoff_ER7xxx.Beckhoff_ER7xxxEK1122.A_0004_ER7041_1002_0025.WcState.InputToggle <-> WcState/InputToggle
//     PlcTask Inputs/GVL_iXlinker.EtherCAT_Master_ERxxxx.Beckhoff_ER7xxx.Beckhoff_ER7xxxEK1122.A_0004_ER7041_1002_0025.InfoData.AdsAddr <-> InfoData/AdsAddr
//     PlcTask Inputs/GVL_iXlinker.EtherCAT_Master_ERxxxx.Beckhoff_ER7xxx.Beckhoff_ER7xxxEK1122.A_0004_ER7041_1002_0025.InfoData.Chn0 <-> InfoData/Chn0
//     PlcTask Inputs/GVL_iXlinker.EtherCAT_Master_ERxxxx.Beckhoff_ER7xxx.Beckhoff_ER7xxxEK1122.A_0004_ER7041_1002_0025.InfoData.Chn1 <-> InfoData/Chn1
//     PlcTask Inputs/GVL_iXlinker.EtherCAT_Master_ERxxxx.Beckhoff_ER7xxx.Beckhoff_ER7xxxEK1122.A_0004_ER7041_1002_0025.InfoData.State <-> InfoData/State
//   PLC/PLC Instance <-> EtherCAT Master ERxxxx/Beckhoff ER7xxx/Beckhoff ER7xxxEK1122/A_0005(ER7041-2002-0024)
//     PlcTask Inputs/GVL_iXlinker.EtherCAT_Master_ERxxxx.Beckhoff_ER7xxx.Beckhoff_ER7xxxEK1122.A_0005_ER7041_2002_0024.ENC_Status_compact.Status/Latch_C_valid <-> ENC Status compact/Status/Latch C valid
//     PlcTask Inputs/GVL_iXlinker.EtherCAT_Master_ERxxxx.Beckhoff_ER7xxx.Beckhoff_ER7xxxEK1122.A_0005_ER7041_2002_0024.ENC_Status_compact.Status/Latch_extern_valid <-> ENC Status compact/Status/Latch extern valid
//     PlcTask Inputs/GVL_iXlinker.EtherCAT_Master_ERxxxx.Beckhoff_ER7xxx.Beckhoff_ER7xxxEK1122.A_0005_ER7041_2002_0024.ENC_Status_compact.Status/Set_counter_done <-> ENC Status compact/Status/Set counter done
//     PlcTask Inputs/GVL_iXlinker.EtherCAT_Master_ERxxxx.Beckhoff_ER7xxx.Beckhoff_ER7xxxEK1122.A_0005_ER7041_2002_0024.ENC_Status_compact.Status/Counter_underflow <-> ENC Status compact/Status/Counter underflow
//     PlcTask Inputs/GVL_iXlinker.EtherCAT_Master_ERxxxx.Beckhoff_ER7xxx.Beckhoff_ER7xxxEK1122.A_0005_ER7041_2002_0024.ENC_Status_compact.Status/Counter_overflow <-> ENC Status compact/Status/Counter overflow
//     PlcTask Inputs/GVL_iXlinker.EtherCAT_Master_ERxxxx.Beckhoff_ER7xxx.Beckhoff_ER7xxxEK1122.A_0005_ER7041_2002_0024.ENC_Status_compact.Status/Extrapolation_stall <-> ENC Status compact/Status/Extrapolation stall
//     PlcTask Inputs/GVL_iXlinker.EtherCAT_Master_ERxxxx.Beckhoff_ER7xxx.Beckhoff_ER7xxxEK1122.A_0005_ER7041_2002_0024.ENC_Status_compact.Status/Status_of_input_A <-> ENC Status compact/Status/Status of input A
//     PlcTask Inputs/GVL_iXlinker.EtherCAT_Master_ERxxxx.Beckhoff_ER7xxx.Beckhoff_ER7xxxEK1122.A_0005_ER7041_2002_0024.ENC_Status_compact.Status/Status_of_input_B <-> ENC Status compact/Status/Status of input B
//     PlcTask Inputs/GVL_iXlinker.EtherCAT_Master_ERxxxx.Beckhoff_ER7xxx.Beckhoff_ER7xxxEK1122.A_0005_ER7041_2002_0024.ENC_Status_compact.Status/Status_of_input_C <-> ENC Status compact/Status/Status of input C
//     PlcTask Inputs/GVL_iXlinker.EtherCAT_Master_ERxxxx.Beckhoff_ER7xxx.Beckhoff_ER7xxxEK1122.A_0005_ER7041_2002_0024.ENC_Status_compact.Status/Status_of_extern_latch <-> ENC Status compact/Status/Status of extern latch
//     PlcTask Inputs/GVL_iXlinker.EtherCAT_Master_ERxxxx.Beckhoff_ER7xxx.Beckhoff_ER7xxxEK1122.A_0005_ER7041_2002_0024.ENC_Status_compact.Status/Sync_error <-> ENC Status compact/Status/Sync error
//     PlcTask Inputs/GVL_iXlinker.EtherCAT_Master_ERxxxx.Beckhoff_ER7xxx.Beckhoff_ER7xxxEK1122.A_0005_ER7041_2002_0024.ENC_Status_compact.Status/TxPDO_Toggle <-> ENC Status compact/Status/TxPDO Toggle
//     PlcTask Inputs/GVL_iXlinker.EtherCAT_Master_ERxxxx.Beckhoff_ER7xxx.Beckhoff_ER7xxxEK1122.A_0005_ER7041_2002_0024.ENC_Status_compact.Counter_value <-> ENC Status compact/Counter value
//     PlcTask Inputs/GVL_iXlinker.EtherCAT_Master_ERxxxx.Beckhoff_ER7xxx.Beckhoff_ER7xxxEK1122.A_0005_ER7041_2002_0024.ENC_Status_compact.Latch_value <-> ENC Status compact/Latch value
//     PlcTask Inputs/GVL_iXlinker.EtherCAT_Master_ERxxxx.Beckhoff_ER7xxx.Beckhoff_ER7xxxEK1122.A_0005_ER7041_2002_0024.STM_Status.Status/Ready_to_enable <-> STM Status/Status/Ready to enable
//     PlcTask Inputs/GVL_iXlinker.EtherCAT_Master_ERxxxx.Beckhoff_ER7xxx.Beckhoff_ER7xxxEK1122.A_0005_ER7041_2002_0024.STM_Status.Status/Ready <-> STM Status/Status/Ready
//     PlcTask Inputs/GVL_iXlinker.EtherCAT_Master_ERxxxx.Beckhoff_ER7xxx.Beckhoff_ER7xxxEK1122.A_0005_ER7041_2002_0024.STM_Status.Status/Warning <-> STM Status/Status/Warning
//     PlcTask Inputs/GVL_iXlinker.EtherCAT_Master_ERxxxx.Beckhoff_ER7xxx.Beckhoff_ER7xxxEK1122.A_0005_ER7041_2002_0024.STM_Status.Status/Error <-> STM Status/Status/Error
//     PlcTask Inputs/GVL_iXlinker.EtherCAT_Master_ERxxxx.Beckhoff_ER7xxx.Beckhoff_ER7xxxEK1122.A_0005_ER7041_2002_0024.STM_Status.Status/Moving_positive <-> STM Status/Status/Moving positive
//     PlcTask Inputs/GVL_iXlinker.EtherCAT_Master_ERxxxx.Beckhoff_ER7xxx.Beckhoff_ER7xxxEK1122.A_0005_ER7041_2002_0024.STM_Status.Status/Moving_negative <-> STM Status/Status/Moving negative
//     PlcTask Inputs/GVL_iXlinker.EtherCAT_Master_ERxxxx.Beckhoff_ER7xxx.Beckhoff_ER7xxxEK1122.A_0005_ER7041_2002_0024.STM_Status.Status/Torque_reduced <-> STM Status/Status/Torque reduced
//     PlcTask Inputs/GVL_iXlinker.EtherCAT_Master_ERxxxx.Beckhoff_ER7xxx.Beckhoff_ER7xxxEK1122.A_0005_ER7041_2002_0024.STM_Status.Status/Digital_input_1 <-> STM Status/Status/Digital input 1
//     PlcTask Inputs/GVL_iXlinker.EtherCAT_Master_ERxxxx.Beckhoff_ER7xxx.Beckhoff_ER7xxxEK1122.A_0005_ER7041_2002_0024.STM_Status.Status/Digital_input_2 <-> STM Status/Status/Digital input 2
//     PlcTask Inputs/GVL_iXlinker.EtherCAT_Master_ERxxxx.Beckhoff_ER7xxx.Beckhoff_ER7xxxEK1122.A_0005_ER7041_2002_0024.STM_Status.Status/Sync_error <-> STM Status/Status/Sync error
//     PlcTask Inputs/GVL_iXlinker.EtherCAT_Master_ERxxxx.Beckhoff_ER7xxx.Beckhoff_ER7xxxEK1122.A_0005_ER7041_2002_0024.STM_Status.Status/TxPDO_Toggle <-> STM Status/Status/TxPDO Toggle
//     PlcTask Outputs/GVL_iXlinker.EtherCAT_Master_ERxxxx.Beckhoff_ER7xxx.Beckhoff_ER7xxxEK1122.A_0005_ER7041_2002_0024.ENC_Control_compact.Control/Enable_latch_C <-> ENC Control compact/Control/Enable latch C
//     PlcTask Outputs/GVL_iXlinker.EtherCAT_Master_ERxxxx.Beckhoff_ER7xxx.Beckhoff_ER7xxxEK1122.A_0005_ER7041_2002_0024.ENC_Control_compact.Control/Enable_latch_extern_on_positive_edge <-> ENC Control compact/Control/Enable latch extern on positive edge
//     PlcTask Outputs/GVL_iXlinker.EtherCAT_Master_ERxxxx.Beckhoff_ER7xxx.Beckhoff_ER7xxxEK1122.A_0005_ER7041_2002_0024.ENC_Control_compact.Control/Set_counter <-> ENC Control compact/Control/Set counter
//     PlcTask Outputs/GVL_iXlinker.EtherCAT_Master_ERxxxx.Beckhoff_ER7xxx.Beckhoff_ER7xxxEK1122.A_0005_ER7041_2002_0024.ENC_Control_compact.Control/Enable_latch_extern_on_negative_edge <-> ENC Control compact/Control/Enable latch extern on negative edge
//     PlcTask Outputs/GVL_iXlinker.EtherCAT_Master_ERxxxx.Beckhoff_ER7xxx.Beckhoff_ER7xxxEK1122.A_0005_ER7041_2002_0024.ENC_Control_compact.Set_counter_value <-> ENC Control compact/Set counter value
//     PlcTask Outputs/GVL_iXlinker.EtherCAT_Master_ERxxxx.Beckhoff_ER7xxx.Beckhoff_ER7xxxEK1122.A_0005_ER7041_2002_0024.STM_Control.Control/Enable <-> STM Control/Control/Enable
//     PlcTask Outputs/GVL_iXlinker.EtherCAT_Master_ERxxxx.Beckhoff_ER7xxx.Beckhoff_ER7xxxEK1122.A_0005_ER7041_2002_0024.STM_Control.Control/Reset <-> STM Control/Control/Reset
//     PlcTask Outputs/GVL_iXlinker.EtherCAT_Master_ERxxxx.Beckhoff_ER7xxx.Beckhoff_ER7xxxEK1122.A_0005_ER7041_2002_0024.STM_Control.Control/Reduce_torque <-> STM Control/Control/Reduce torque
//     PlcTask Outputs/GVL_iXlinker.EtherCAT_Master_ERxxxx.Beckhoff_ER7xxx.Beckhoff_ER7xxxEK1122.A_0005_ER7041_2002_0024.STM_Control.Control/Digital_output_1 <-> STM Control/Control/Digital output 1
//     PlcTask Outputs/GVL_iXlinker.EtherCAT_Master_ERxxxx.Beckhoff_ER7xxx.Beckhoff_ER7xxxEK1122.A_0005_ER7041_2002_0024.STM_Velocity.Velocity <-> STM Velocity/Velocity
//     PlcTask Inputs/GVL_iXlinker.EtherCAT_Master_ERxxxx.Beckhoff_ER7xxx.Beckhoff_ER7xxxEK1122.A_0005_ER7041_2002_0024.WcState.WcState <-> WcState/WcState
//     PlcTask Inputs/GVL_iXlinker.EtherCAT_Master_ERxxxx.Beckhoff_ER7xxx.Beckhoff_ER7xxxEK1122.A_0005_ER7041_2002_0024.WcState.InputToggle <-> WcState/InputToggle
//     PlcTask Inputs/GVL_iXlinker.EtherCAT_Master_ERxxxx.Beckhoff_ER7xxx.Beckhoff_ER7xxxEK1122.A_0005_ER7041_2002_0024.InfoData.AdsAddr <-> InfoData/AdsAddr
//     PlcTask Inputs/GVL_iXlinker.EtherCAT_Master_ERxxxx.Beckhoff_ER7xxx.Beckhoff_ER7xxxEK1122.A_0005_ER7041_2002_0024.InfoData.Chn0 <-> InfoData/Chn0
//     PlcTask Inputs/GVL_iXlinker.EtherCAT_Master_ERxxxx.Beckhoff_ER7xxx.Beckhoff_ER7xxxEK1122.A_0005_ER7041_2002_0024.InfoData.Chn1 <-> InfoData/Chn1
//     PlcTask Inputs/GVL_iXlinker.EtherCAT_Master_ERxxxx.Beckhoff_ER7xxx.Beckhoff_ER7xxxEK1122.A_0005_ER7041_2002_0024.InfoData.State <-> InfoData/State
//   PLC/PLC Instance <-> EtherCAT Master ERxxxx/Beckhoff ER7xxx/Beckhoff ER7xxxEK1122/A_0006(ER7041-2002-0025)
//     PlcTask Inputs/GVL_iXlinker.EtherCAT_Master_ERxxxx.Beckhoff_ER7xxx.Beckhoff_ER7xxxEK1122.A_0006_ER7041_2002_0025.ENC_Status_compact.Status/Latch_C_valid <-> ENC Status compact/Status/Latch C valid
//     PlcTask Inputs/GVL_iXlinker.EtherCAT_Master_ERxxxx.Beckhoff_ER7xxx.Beckhoff_ER7xxxEK1122.A_0006_ER7041_2002_0025.ENC_Status_compact.Status/Latch_extern_valid <-> ENC Status compact/Status/Latch extern valid
//     PlcTask Inputs/GVL_iXlinker.EtherCAT_Master_ERxxxx.Beckhoff_ER7xxx.Beckhoff_ER7xxxEK1122.A_0006_ER7041_2002_0025.ENC_Status_compact.Status/Set_counter_done <-> ENC Status compact/Status/Set counter done
//     PlcTask Inputs/GVL_iXlinker.EtherCAT_Master_ERxxxx.Beckhoff_ER7xxx.Beckhoff_ER7xxxEK1122.A_0006_ER7041_2002_0025.ENC_Status_compact.Status/Counter_underflow <-> ENC Status compact/Status/Counter underflow
//     PlcTask Inputs/GVL_iXlinker.EtherCAT_Master_ERxxxx.Beckhoff_ER7xxx.Beckhoff_ER7xxxEK1122.A_0006_ER7041_2002_0025.ENC_Status_compact.Status/Counter_overflow <-> ENC Status compact/Status/Counter overflow
//     PlcTask Inputs/GVL_iXlinker.EtherCAT_Master_ERxxxx.Beckhoff_ER7xxx.Beckhoff_ER7xxxEK1122.A_0006_ER7041_2002_0025.ENC_Status_compact.Status/Extrapolation_stall <-> ENC Status compact/Status/Extrapolation stall
//     PlcTask Inputs/GVL_iXlinker.EtherCAT_Master_ERxxxx.Beckhoff_ER7xxx.Beckhoff_ER7xxxEK1122.A_0006_ER7041_2002_0025.ENC_Status_compact.Status/Status_of_input_A <-> ENC Status compact/Status/Status of input A
//     PlcTask Inputs/GVL_iXlinker.EtherCAT_Master_ERxxxx.Beckhoff_ER7xxx.Beckhoff_ER7xxxEK1122.A_0006_ER7041_2002_0025.ENC_Status_compact.Status/Status_of_input_B <-> ENC Status compact/Status/Status of input B
//     PlcTask Inputs/GVL_iXlinker.EtherCAT_Master_ERxxxx.Beckhoff_ER7xxx.Beckhoff_ER7xxxEK1122.A_0006_ER7041_2002_0025.ENC_Status_compact.Status/Status_of_input_C <-> ENC Status compact/Status/Status of input C
//     PlcTask Inputs/GVL_iXlinker.EtherCAT_Master_ERxxxx.Beckhoff_ER7xxx.Beckhoff_ER7xxxEK1122.A_0006_ER7041_2002_0025.ENC_Status_compact.Status/Status_of_extern_latch <-> ENC Status compact/Status/Status of extern latch
//     PlcTask Inputs/GVL_iXlinker.EtherCAT_Master_ERxxxx.Beckhoff_ER7xxx.Beckhoff_ER7xxxEK1122.A_0006_ER7041_2002_0025.ENC_Status_compact.Status/Sync_error <-> ENC Status compact/Status/Sync error
//     PlcTask Inputs/GVL_iXlinker.EtherCAT_Master_ERxxxx.Beckhoff_ER7xxx.Beckhoff_ER7xxxEK1122.A_0006_ER7041_2002_0025.ENC_Status_compact.Status/TxPDO_Toggle <-> ENC Status compact/Status/TxPDO Toggle
//     PlcTask Inputs/GVL_iXlinker.EtherCAT_Master_ERxxxx.Beckhoff_ER7xxx.Beckhoff_ER7xxxEK1122.A_0006_ER7041_2002_0025.ENC_Status_compact.Counter_value <-> ENC Status compact/Counter value
//     PlcTask Inputs/GVL_iXlinker.EtherCAT_Master_ERxxxx.Beckhoff_ER7xxx.Beckhoff_ER7xxxEK1122.A_0006_ER7041_2002_0025.ENC_Status_compact.Latch_value <-> ENC Status compact/Latch value
//     PlcTask Inputs/GVL_iXlinker.EtherCAT_Master_ERxxxx.Beckhoff_ER7xxx.Beckhoff_ER7xxxEK1122.A_0006_ER7041_2002_0025.STM_Status.Status/Ready_to_enable <-> STM Status/Status/Ready to enable
//     PlcTask Inputs/GVL_iXlinker.EtherCAT_Master_ERxxxx.Beckhoff_ER7xxx.Beckhoff_ER7xxxEK1122.A_0006_ER7041_2002_0025.STM_Status.Status/Ready <-> STM Status/Status/Ready
//     PlcTask Inputs/GVL_iXlinker.EtherCAT_Master_ERxxxx.Beckhoff_ER7xxx.Beckhoff_ER7xxxEK1122.A_0006_ER7041_2002_0025.STM_Status.Status/Warning <-> STM Status/Status/Warning
//     PlcTask Inputs/GVL_iXlinker.EtherCAT_Master_ERxxxx.Beckhoff_ER7xxx.Beckhoff_ER7xxxEK1122.A_0006_ER7041_2002_0025.STM_Status.Status/Error <-> STM Status/Status/Error
//     PlcTask Inputs/GVL_iXlinker.EtherCAT_Master_ERxxxx.Beckhoff_ER7xxx.Beckhoff_ER7xxxEK1122.A_0006_ER7041_2002_0025.STM_Status.Status/Moving_positive <-> STM Status/Status/Moving positive
//     PlcTask Inputs/GVL_iXlinker.EtherCAT_Master_ERxxxx.Beckhoff_ER7xxx.Beckhoff_ER7xxxEK1122.A_0006_ER7041_2002_0025.STM_Status.Status/Moving_negative <-> STM Status/Status/Moving negative
//     PlcTask Inputs/GVL_iXlinker.EtherCAT_Master_ERxxxx.Beckhoff_ER7xxx.Beckhoff_ER7xxxEK1122.A_0006_ER7041_2002_0025.STM_Status.Status/Torque_reduced <-> STM Status/Status/Torque reduced
//     PlcTask Inputs/GVL_iXlinker.EtherCAT_Master_ERxxxx.Beckhoff_ER7xxx.Beckhoff_ER7xxxEK1122.A_0006_ER7041_2002_0025.STM_Status.Status/Digital_input_1 <-> STM Status/Status/Digital input 1
//     PlcTask Inputs/GVL_iXlinker.EtherCAT_Master_ERxxxx.Beckhoff_ER7xxx.Beckhoff_ER7xxxEK1122.A_0006_ER7041_2002_0025.STM_Status.Status/Digital_input_2 <-> STM Status/Status/Digital input 2
//     PlcTask Inputs/GVL_iXlinker.EtherCAT_Master_ERxxxx.Beckhoff_ER7xxx.Beckhoff_ER7xxxEK1122.A_0006_ER7041_2002_0025.STM_Status.Status/Sync_error <-> STM Status/Status/Sync error
//     PlcTask Inputs/GVL_iXlinker.EtherCAT_Master_ERxxxx.Beckhoff_ER7xxx.Beckhoff_ER7xxxEK1122.A_0006_ER7041_2002_0025.STM_Status.Status/TxPDO_Toggle <-> STM Status/Status/TxPDO Toggle
//     PlcTask Outputs/GVL_iXlinker.EtherCAT_Master_ERxxxx.Beckhoff_ER7xxx.Beckhoff_ER7xxxEK1122.A_0006_ER7041_2002_0025.ENC_Control_compact.Control/Enable_latch_C <-> ENC Control compact/Control/Enable latch C
//     PlcTask Outputs/GVL_iXlinker.EtherCAT_Master_ERxxxx.Beckhoff_ER7xxx.Beckhoff_ER7xxxEK1122.A_0006_ER7041_2002_0025.ENC_Control_compact.Control/Enable_latch_extern_on_positive_edge <-> ENC Control compact/Control/Enable latch extern on positive edge
//     PlcTask Outputs/GVL_iXlinker.EtherCAT_Master_ERxxxx.Beckhoff_ER7xxx.Beckhoff_ER7xxxEK1122.A_0006_ER7041_2002_0025.ENC_Control_compact.Control/Set_counter <-> ENC Control compact/Control/Set counter
//     PlcTask Outputs/GVL_iXlinker.EtherCAT_Master_ERxxxx.Beckhoff_ER7xxx.Beckhoff_ER7xxxEK1122.A_0006_ER7041_2002_0025.ENC_Control_compact.Control/Enable_latch_extern_on_negative_edge <-> ENC Control compact/Control/Enable latch extern on negative edge
//     PlcTask Outputs/GVL_iXlinker.EtherCAT_Master_ERxxxx.Beckhoff_ER7xxx.Beckhoff_ER7xxxEK1122.A_0006_ER7041_2002_0025.ENC_Control_compact.Set_counter_value <-> ENC Control compact/Set counter value
//     PlcTask Outputs/GVL_iXlinker.EtherCAT_Master_ERxxxx.Beckhoff_ER7xxx.Beckhoff_ER7xxxEK1122.A_0006_ER7041_2002_0025.STM_Control.Control/Enable <-> STM Control/Control/Enable
//     PlcTask Outputs/GVL_iXlinker.EtherCAT_Master_ERxxxx.Beckhoff_ER7xxx.Beckhoff_ER7xxxEK1122.A_0006_ER7041_2002_0025.STM_Control.Control/Reset <-> STM Control/Control/Reset
//     PlcTask Outputs/GVL_iXlinker.EtherCAT_Master_ERxxxx.Beckhoff_ER7xxx.Beckhoff_ER7xxxEK1122.A_0006_ER7041_2002_0025.STM_Control.Control/Reduce_torque <-> STM Control/Control/Reduce torque
//     PlcTask Outputs/GVL_iXlinker.EtherCAT_Master_ERxxxx.Beckhoff_ER7xxx.Beckhoff_ER7xxxEK1122.A_0006_ER7041_2002_0025.STM_Control.Control/Digital_output_1 <-> STM Control/Control/Digital output 1
//     PlcTask Outputs/GVL_iXlinker.EtherCAT_Master_ERxxxx.Beckhoff_ER7xxx.Beckhoff_ER7xxxEK1122.A_0006_ER7041_2002_0025.STM_Velocity.Velocity <-> STM Velocity/Velocity
//     PlcTask Inputs/GVL_iXlinker.EtherCAT_Master_ERxxxx.Beckhoff_ER7xxx.Beckhoff_ER7xxxEK1122.A_0006_ER7041_2002_0025.WcState.WcState <-> WcState/WcState
//     PlcTask Inputs/GVL_iXlinker.EtherCAT_Master_ERxxxx.Beckhoff_ER7xxx.Beckhoff_ER7xxxEK1122.A_0006_ER7041_2002_0025.WcState.InputToggle <-> WcState/InputToggle
//     PlcTask Inputs/GVL_iXlinker.EtherCAT_Master_ERxxxx.Beckhoff_ER7xxx.Beckhoff_ER7xxxEK1122.A_0006_ER7041_2002_0025.InfoData.AdsAddr <-> InfoData/AdsAddr
//     PlcTask Inputs/GVL_iXlinker.EtherCAT_Master_ERxxxx.Beckhoff_ER7xxx.Beckhoff_ER7xxxEK1122.A_0006_ER7041_2002_0025.InfoData.Chn0 <-> InfoData/Chn0
//     PlcTask Inputs/GVL_iXlinker.EtherCAT_Master_ERxxxx.Beckhoff_ER7xxx.Beckhoff_ER7xxxEK1122.A_0006_ER7041_2002_0025.InfoData.Chn1 <-> InfoData/Chn1
//     PlcTask Inputs/GVL_iXlinker.EtherCAT_Master_ERxxxx.Beckhoff_ER7xxx.Beckhoff_ER7xxxEK1122.A_0006_ER7041_2002_0025.InfoData.State <-> InfoData/State
//   PLC/PLC Instance <-> EtherCAT Master ERxxxx/Beckhoff ER7xxx/Beckhoff ER7xxxEK1122/A_0007(ER7041-3002-0021)
//     PlcTask Inputs/GVL_iXlinker.EtherCAT_Master_ERxxxx.Beckhoff_ER7xxx.Beckhoff_ER7xxxEK1122.A_0007_ER7041_3002_0021.ENC_Status_compact.Status/Latch_C_valid <-> ENC Status compact/Status/Latch C valid
//     PlcTask Inputs/GVL_iXlinker.EtherCAT_Master_ERxxxx.Beckhoff_ER7xxx.Beckhoff_ER7xxxEK1122.A_0007_ER7041_3002_0021.ENC_Status_compact.Status/Latch_extern_valid <-> ENC Status compact/Status/Latch extern valid
//     PlcTask Inputs/GVL_iXlinker.EtherCAT_Master_ERxxxx.Beckhoff_ER7xxx.Beckhoff_ER7xxxEK1122.A_0007_ER7041_3002_0021.ENC_Status_compact.Status/Set_counter_done <-> ENC Status compact/Status/Set counter done
//     PlcTask Inputs/GVL_iXlinker.EtherCAT_Master_ERxxxx.Beckhoff_ER7xxx.Beckhoff_ER7xxxEK1122.A_0007_ER7041_3002_0021.ENC_Status_compact.Status/Counter_underflow <-> ENC Status compact/Status/Counter underflow
//     PlcTask Inputs/GVL_iXlinker.EtherCAT_Master_ERxxxx.Beckhoff_ER7xxx.Beckhoff_ER7xxxEK1122.A_0007_ER7041_3002_0021.ENC_Status_compact.Status/Counter_overflow <-> ENC Status compact/Status/Counter overflow
//     PlcTask Inputs/GVL_iXlinker.EtherCAT_Master_ERxxxx.Beckhoff_ER7xxx.Beckhoff_ER7xxxEK1122.A_0007_ER7041_3002_0021.ENC_Status_compact.Status/Extrapolation_stall <-> ENC Status compact/Status/Extrapolation stall
//     PlcTask Inputs/GVL_iXlinker.EtherCAT_Master_ERxxxx.Beckhoff_ER7xxx.Beckhoff_ER7xxxEK1122.A_0007_ER7041_3002_0021.ENC_Status_compact.Status/Status_of_input_A <-> ENC Status compact/Status/Status of input A
//     PlcTask Inputs/GVL_iXlinker.EtherCAT_Master_ERxxxx.Beckhoff_ER7xxx.Beckhoff_ER7xxxEK1122.A_0007_ER7041_3002_0021.ENC_Status_compact.Status/Status_of_input_B <-> ENC Status compact/Status/Status of input B
//     PlcTask Inputs/GVL_iXlinker.EtherCAT_Master_ERxxxx.Beckhoff_ER7xxx.Beckhoff_ER7xxxEK1122.A_0007_ER7041_3002_0021.ENC_Status_compact.Status/Status_of_input_C <-> ENC Status compact/Status/Status of input C
//     PlcTask Inputs/GVL_iXlinker.EtherCAT_Master_ERxxxx.Beckhoff_ER7xxx.Beckhoff_ER7xxxEK1122.A_0007_ER7041_3002_0021.ENC_Status_compact.Status/Status_of_extern_latch <-> ENC Status compact/Status/Status of extern latch
//     PlcTask Inputs/GVL_iXlinker.EtherCAT_Master_ERxxxx.Beckhoff_ER7xxx.Beckhoff_ER7xxxEK1122.A_0007_ER7041_3002_0021.ENC_Status_compact.Status/Sync_error <-> ENC Status compact/Status/Sync error
//     PlcTask Inputs/GVL_iXlinker.EtherCAT_Master_ERxxxx.Beckhoff_ER7xxx.Beckhoff_ER7xxxEK1122.A_0007_ER7041_3002_0021.ENC_Status_compact.Status/TxPDO_Toggle <-> ENC Status compact/Status/TxPDO Toggle
//     PlcTask Inputs/GVL_iXlinker.EtherCAT_Master_ERxxxx.Beckhoff_ER7xxx.Beckhoff_ER7xxxEK1122.A_0007_ER7041_3002_0021.ENC_Status_compact.Counter_value <-> ENC Status compact/Counter value
//     PlcTask Inputs/GVL_iXlinker.EtherCAT_Master_ERxxxx.Beckhoff_ER7xxx.Beckhoff_ER7xxxEK1122.A_0007_ER7041_3002_0021.ENC_Status_compact.Latch_value <-> ENC Status compact/Latch value
//     PlcTask Inputs/GVL_iXlinker.EtherCAT_Master_ERxxxx.Beckhoff_ER7xxx.Beckhoff_ER7xxxEK1122.A_0007_ER7041_3002_0021.STM_Status.Status/Ready_to_enable <-> STM Status/Status/Ready to enable
//     PlcTask Inputs/GVL_iXlinker.EtherCAT_Master_ERxxxx.Beckhoff_ER7xxx.Beckhoff_ER7xxxEK1122.A_0007_ER7041_3002_0021.STM_Status.Status/Ready <-> STM Status/Status/Ready
//     PlcTask Inputs/GVL_iXlinker.EtherCAT_Master_ERxxxx.Beckhoff_ER7xxx.Beckhoff_ER7xxxEK1122.A_0007_ER7041_3002_0021.STM_Status.Status/Warning <-> STM Status/Status/Warning
//     PlcTask Inputs/GVL_iXlinker.EtherCAT_Master_ERxxxx.Beckhoff_ER7xxx.Beckhoff_ER7xxxEK1122.A_0007_ER7041_3002_0021.STM_Status.Status/Error <-> STM Status/Status/Error
//     PlcTask Inputs/GVL_iXlinker.EtherCAT_Master_ERxxxx.Beckhoff_ER7xxx.Beckhoff_ER7xxxEK1122.A_0007_ER7041_3002_0021.STM_Status.Status/Moving_positive <-> STM Status/Status/Moving positive
//     PlcTask Inputs/GVL_iXlinker.EtherCAT_Master_ERxxxx.Beckhoff_ER7xxx.Beckhoff_ER7xxxEK1122.A_0007_ER7041_3002_0021.STM_Status.Status/Moving_negative <-> STM Status/Status/Moving negative
//     PlcTask Inputs/GVL_iXlinker.EtherCAT_Master_ERxxxx.Beckhoff_ER7xxx.Beckhoff_ER7xxxEK1122.A_0007_ER7041_3002_0021.STM_Status.Status/Torque_reduced <-> STM Status/Status/Torque reduced
//     PlcTask Inputs/GVL_iXlinker.EtherCAT_Master_ERxxxx.Beckhoff_ER7xxx.Beckhoff_ER7xxxEK1122.A_0007_ER7041_3002_0021.STM_Status.Status/Motor_stall <-> STM Status/Status/Motor stall
//     PlcTask Inputs/GVL_iXlinker.EtherCAT_Master_ERxxxx.Beckhoff_ER7xxx.Beckhoff_ER7xxxEK1122.A_0007_ER7041_3002_0021.STM_Status.Status/Digital_input_1 <-> STM Status/Status/Digital input 1
//     PlcTask Inputs/GVL_iXlinker.EtherCAT_Master_ERxxxx.Beckhoff_ER7xxx.Beckhoff_ER7xxxEK1122.A_0007_ER7041_3002_0021.STM_Status.Status/Digital_input_2 <-> STM Status/Status/Digital input 2
//     PlcTask Inputs/GVL_iXlinker.EtherCAT_Master_ERxxxx.Beckhoff_ER7xxx.Beckhoff_ER7xxxEK1122.A_0007_ER7041_3002_0021.STM_Status.Status/Sync_error <-> STM Status/Status/Sync error
//     PlcTask Inputs/GVL_iXlinker.EtherCAT_Master_ERxxxx.Beckhoff_ER7xxx.Beckhoff_ER7xxxEK1122.A_0007_ER7041_3002_0021.STM_Status.Status/TxPDO_Toggle <-> STM Status/Status/TxPDO Toggle
//     PlcTask Outputs/GVL_iXlinker.EtherCAT_Master_ERxxxx.Beckhoff_ER7xxx.Beckhoff_ER7xxxEK1122.A_0007_ER7041_3002_0021.ENC_Control_compact.Control/Enable_latch_C <-> ENC Control compact/Control/Enable latch C
//     PlcTask Outputs/GVL_iXlinker.EtherCAT_Master_ERxxxx.Beckhoff_ER7xxx.Beckhoff_ER7xxxEK1122.A_0007_ER7041_3002_0021.ENC_Control_compact.Control/Enable_latch_extern_on_positive_edge <-> ENC Control compact/Control/Enable latch extern on positive edge
//     PlcTask Outputs/GVL_iXlinker.EtherCAT_Master_ERxxxx.Beckhoff_ER7xxx.Beckhoff_ER7xxxEK1122.A_0007_ER7041_3002_0021.ENC_Control_compact.Control/Set_counter <-> ENC Control compact/Control/Set counter
//     PlcTask Outputs/GVL_iXlinker.EtherCAT_Master_ERxxxx.Beckhoff_ER7xxx.Beckhoff_ER7xxxEK1122.A_0007_ER7041_3002_0021.ENC_Control_compact.Control/Enable_latch_extern_on_negative_edge <-> ENC Control compact/Control/Enable latch extern on negative edge
//     PlcTask Outputs/GVL_iXlinker.EtherCAT_Master_ERxxxx.Beckhoff_ER7xxx.Beckhoff_ER7xxxEK1122.A_0007_ER7041_3002_0021.ENC_Control_compact.Set_counter_value <-> ENC Control compact/Set counter value
//     PlcTask Outputs/GVL_iXlinker.EtherCAT_Master_ERxxxx.Beckhoff_ER7xxx.Beckhoff_ER7xxxEK1122.A_0007_ER7041_3002_0021.STM_Control.Control/Enable <-> STM Control/Control/Enable
//     PlcTask Outputs/GVL_iXlinker.EtherCAT_Master_ERxxxx.Beckhoff_ER7xxx.Beckhoff_ER7xxxEK1122.A_0007_ER7041_3002_0021.STM_Control.Control/Reset <-> STM Control/Control/Reset
//     PlcTask Outputs/GVL_iXlinker.EtherCAT_Master_ERxxxx.Beckhoff_ER7xxx.Beckhoff_ER7xxxEK1122.A_0007_ER7041_3002_0021.STM_Control.Control/Reduce_torque <-> STM Control/Control/Reduce torque
//     PlcTask Outputs/GVL_iXlinker.EtherCAT_Master_ERxxxx.Beckhoff_ER7xxx.Beckhoff_ER7xxxEK1122.A_0007_ER7041_3002_0021.STM_Control.Control/Digital_output_1 <-> STM Control/Control/Digital output 1
//     PlcTask Outputs/GVL_iXlinker.EtherCAT_Master_ERxxxx.Beckhoff_ER7xxx.Beckhoff_ER7xxxEK1122.A_0007_ER7041_3002_0021.STM_Velocity.Velocity <-> STM Velocity/Velocity
//     PlcTask Inputs/GVL_iXlinker.EtherCAT_Master_ERxxxx.Beckhoff_ER7xxx.Beckhoff_ER7xxxEK1122.A_0007_ER7041_3002_0021.WcState.WcState <-> WcState/WcState
//     PlcTask Inputs/GVL_iXlinker.EtherCAT_Master_ERxxxx.Beckhoff_ER7xxx.Beckhoff_ER7xxxEK1122.A_0007_ER7041_3002_0021.WcState.InputToggle <-> WcState/InputToggle
//     PlcTask Inputs/GVL_iXlinker.EtherCAT_Master_ERxxxx.Beckhoff_ER7xxx.Beckhoff_ER7xxxEK1122.A_0007_ER7041_3002_0021.InfoData.AdsAddr <-> InfoData/AdsAddr
//     PlcTask Inputs/GVL_iXlinker.EtherCAT_Master_ERxxxx.Beckhoff_ER7xxx.Beckhoff_ER7xxxEK1122.A_0007_ER7041_3002_0021.InfoData.Chn0 <-> InfoData/Chn0
//     PlcTask Inputs/GVL_iXlinker.EtherCAT_Master_ERxxxx.Beckhoff_ER7xxx.Beckhoff_ER7xxxEK1122.A_0007_ER7041_3002_0021.InfoData.Chn1 <-> InfoData/Chn1
//     PlcTask Inputs/GVL_iXlinker.EtherCAT_Master_ERxxxx.Beckhoff_ER7xxx.Beckhoff_ER7xxxEK1122.A_0007_ER7041_3002_0021.InfoData.State <-> InfoData/State
//   PLC/PLC Instance <-> EtherCAT Master ERxxxx/Beckhoff ER7xxx/Beckhoff ER7xxxEK1122/A_0008(ER7041-3002-0022)
//     PlcTask Inputs/GVL_iXlinker.EtherCAT_Master_ERxxxx.Beckhoff_ER7xxx.Beckhoff_ER7xxxEK1122.A_0008_ER7041_3002_0022.ENC_Status_compact.Status/Latch_C_valid <-> ENC Status compact/Status/Latch C valid
//     PlcTask Inputs/GVL_iXlinker.EtherCAT_Master_ERxxxx.Beckhoff_ER7xxx.Beckhoff_ER7xxxEK1122.A_0008_ER7041_3002_0022.ENC_Status_compact.Status/Latch_extern_valid <-> ENC Status compact/Status/Latch extern valid
//     PlcTask Inputs/GVL_iXlinker.EtherCAT_Master_ERxxxx.Beckhoff_ER7xxx.Beckhoff_ER7xxxEK1122.A_0008_ER7041_3002_0022.ENC_Status_compact.Status/Set_counter_done <-> ENC Status compact/Status/Set counter done
//     PlcTask Inputs/GVL_iXlinker.EtherCAT_Master_ERxxxx.Beckhoff_ER7xxx.Beckhoff_ER7xxxEK1122.A_0008_ER7041_3002_0022.ENC_Status_compact.Status/Counter_underflow <-> ENC Status compact/Status/Counter underflow
//     PlcTask Inputs/GVL_iXlinker.EtherCAT_Master_ERxxxx.Beckhoff_ER7xxx.Beckhoff_ER7xxxEK1122.A_0008_ER7041_3002_0022.ENC_Status_compact.Status/Counter_overflow <-> ENC Status compact/Status/Counter overflow
//     PlcTask Inputs/GVL_iXlinker.EtherCAT_Master_ERxxxx.Beckhoff_ER7xxx.Beckhoff_ER7xxxEK1122.A_0008_ER7041_3002_0022.ENC_Status_compact.Status/Extrapolation_stall <-> ENC Status compact/Status/Extrapolation stall
//     PlcTask Inputs/GVL_iXlinker.EtherCAT_Master_ERxxxx.Beckhoff_ER7xxx.Beckhoff_ER7xxxEK1122.A_0008_ER7041_3002_0022.ENC_Status_compact.Status/Status_of_input_A <-> ENC Status compact/Status/Status of input A
//     PlcTask Inputs/GVL_iXlinker.EtherCAT_Master_ERxxxx.Beckhoff_ER7xxx.Beckhoff_ER7xxxEK1122.A_0008_ER7041_3002_0022.ENC_Status_compact.Status/Status_of_input_B <-> ENC Status compact/Status/Status of input B
//     PlcTask Inputs/GVL_iXlinker.EtherCAT_Master_ERxxxx.Beckhoff_ER7xxx.Beckhoff_ER7xxxEK1122.A_0008_ER7041_3002_0022.ENC_Status_compact.Status/Status_of_input_C <-> ENC Status compact/Status/Status of input C
//     PlcTask Inputs/GVL_iXlinker.EtherCAT_Master_ERxxxx.Beckhoff_ER7xxx.Beckhoff_ER7xxxEK1122.A_0008_ER7041_3002_0022.ENC_Status_compact.Status/Status_of_extern_latch <-> ENC Status compact/Status/Status of extern latch
//     PlcTask Inputs/GVL_iXlinker.EtherCAT_Master_ERxxxx.Beckhoff_ER7xxx.Beckhoff_ER7xxxEK1122.A_0008_ER7041_3002_0022.ENC_Status_compact.Status/Sync_error <-> ENC Status compact/Status/Sync error
//     PlcTask Inputs/GVL_iXlinker.EtherCAT_Master_ERxxxx.Beckhoff_ER7xxx.Beckhoff_ER7xxxEK1122.A_0008_ER7041_3002_0022.ENC_Status_compact.Status/TxPDO_Toggle <-> ENC Status compact/Status/TxPDO Toggle
//     PlcTask Inputs/GVL_iXlinker.EtherCAT_Master_ERxxxx.Beckhoff_ER7xxx.Beckhoff_ER7xxxEK1122.A_0008_ER7041_3002_0022.ENC_Status_compact.Counter_value <-> ENC Status compact/Counter value
//     PlcTask Inputs/GVL_iXlinker.EtherCAT_Master_ERxxxx.Beckhoff_ER7xxx.Beckhoff_ER7xxxEK1122.A_0008_ER7041_3002_0022.ENC_Status_compact.Latch_value <-> ENC Status compact/Latch value
//     PlcTask Inputs/GVL_iXlinker.EtherCAT_Master_ERxxxx.Beckhoff_ER7xxx.Beckhoff_ER7xxxEK1122.A_0008_ER7041_3002_0022.STM_Status.Status/Ready_to_enable <-> STM Status/Status/Ready to enable
//     PlcTask Inputs/GVL_iXlinker.EtherCAT_Master_ERxxxx.Beckhoff_ER7xxx.Beckhoff_ER7xxxEK1122.A_0008_ER7041_3002_0022.STM_Status.Status/Ready <-> STM Status/Status/Ready
//     PlcTask Inputs/GVL_iXlinker.EtherCAT_Master_ERxxxx.Beckhoff_ER7xxx.Beckhoff_ER7xxxEK1122.A_0008_ER7041_3002_0022.STM_Status.Status/Warning <-> STM Status/Status/Warning
//     PlcTask Inputs/GVL_iXlinker.EtherCAT_Master_ERxxxx.Beckhoff_ER7xxx.Beckhoff_ER7xxxEK1122.A_0008_ER7041_3002_0022.STM_Status.Status/Error <-> STM Status/Status/Error
//     PlcTask Inputs/GVL_iXlinker.EtherCAT_Master_ERxxxx.Beckhoff_ER7xxx.Beckhoff_ER7xxxEK1122.A_0008_ER7041_3002_0022.STM_Status.Status/Moving_positive <-> STM Status/Status/Moving positive
//     PlcTask Inputs/GVL_iXlinker.EtherCAT_Master_ERxxxx.Beckhoff_ER7xxx.Beckhoff_ER7xxxEK1122.A_0008_ER7041_3002_0022.STM_Status.Status/Moving_negative <-> STM Status/Status/Moving negative
//     PlcTask Inputs/GVL_iXlinker.EtherCAT_Master_ERxxxx.Beckhoff_ER7xxx.Beckhoff_ER7xxxEK1122.A_0008_ER7041_3002_0022.STM_Status.Status/Torque_reduced <-> STM Status/Status/Torque reduced
//     PlcTask Inputs/GVL_iXlinker.EtherCAT_Master_ERxxxx.Beckhoff_ER7xxx.Beckhoff_ER7xxxEK1122.A_0008_ER7041_3002_0022.STM_Status.Status/Motor_stall <-> STM Status/Status/Motor stall
//     PlcTask Inputs/GVL_iXlinker.EtherCAT_Master_ERxxxx.Beckhoff_ER7xxx.Beckhoff_ER7xxxEK1122.A_0008_ER7041_3002_0022.STM_Status.Status/Digital_input_1 <-> STM Status/Status/Digital input 1
//     PlcTask Inputs/GVL_iXlinker.EtherCAT_Master_ERxxxx.Beckhoff_ER7xxx.Beckhoff_ER7xxxEK1122.A_0008_ER7041_3002_0022.STM_Status.Status/Digital_input_2 <-> STM Status/Status/Digital input 2
//     PlcTask Inputs/GVL_iXlinker.EtherCAT_Master_ERxxxx.Beckhoff_ER7xxx.Beckhoff_ER7xxxEK1122.A_0008_ER7041_3002_0022.STM_Status.Status/Sync_error <-> STM Status/Status/Sync error
//     PlcTask Inputs/GVL_iXlinker.EtherCAT_Master_ERxxxx.Beckhoff_ER7xxx.Beckhoff_ER7xxxEK1122.A_0008_ER7041_3002_0022.STM_Status.Status/TxPDO_Toggle <-> STM Status/Status/TxPDO Toggle
//     PlcTask Outputs/GVL_iXlinker.EtherCAT_Master_ERxxxx.Beckhoff_ER7xxx.Beckhoff_ER7xxxEK1122.A_0008_ER7041_3002_0022.ENC_Control_compact.Control/Enable_latch_C <-> ENC Control compact/Control/Enable latch C
//     PlcTask Outputs/GVL_iXlinker.EtherCAT_Master_ERxxxx.Beckhoff_ER7xxx.Beckhoff_ER7xxxEK1122.A_0008_ER7041_3002_0022.ENC_Control_compact.Control/Enable_latch_extern_on_positive_edge <-> ENC Control compact/Control/Enable latch extern on positive edge
//     PlcTask Outputs/GVL_iXlinker.EtherCAT_Master_ERxxxx.Beckhoff_ER7xxx.Beckhoff_ER7xxxEK1122.A_0008_ER7041_3002_0022.ENC_Control_compact.Control/Set_counter <-> ENC Control compact/Control/Set counter
//     PlcTask Outputs/GVL_iXlinker.EtherCAT_Master_ERxxxx.Beckhoff_ER7xxx.Beckhoff_ER7xxxEK1122.A_0008_ER7041_3002_0022.ENC_Control_compact.Control/Enable_latch_extern_on_negative_edge <-> ENC Control compact/Control/Enable latch extern on negative edge
//     PlcTask Outputs/GVL_iXlinker.EtherCAT_Master_ERxxxx.Beckhoff_ER7xxx.Beckhoff_ER7xxxEK1122.A_0008_ER7041_3002_0022.ENC_Control_compact.Set_counter_value <-> ENC Control compact/Set counter value
//     PlcTask Outputs/GVL_iXlinker.EtherCAT_Master_ERxxxx.Beckhoff_ER7xxx.Beckhoff_ER7xxxEK1122.A_0008_ER7041_3002_0022.STM_Control.Control/Enable <-> STM Control/Control/Enable
//     PlcTask Outputs/GVL_iXlinker.EtherCAT_Master_ERxxxx.Beckhoff_ER7xxx.Beckhoff_ER7xxxEK1122.A_0008_ER7041_3002_0022.STM_Control.Control/Reset <-> STM Control/Control/Reset
//     PlcTask Outputs/GVL_iXlinker.EtherCAT_Master_ERxxxx.Beckhoff_ER7xxx.Beckhoff_ER7xxxEK1122.A_0008_ER7041_3002_0022.STM_Control.Control/Reduce_torque <-> STM Control/Control/Reduce torque
//     PlcTask Outputs/GVL_iXlinker.EtherCAT_Master_ERxxxx.Beckhoff_ER7xxx.Beckhoff_ER7xxxEK1122.A_0008_ER7041_3002_0022.STM_Control.Control/Digital_output_1 <-> STM Control/Control/Digital output 1
//     PlcTask Outputs/GVL_iXlinker.EtherCAT_Master_ERxxxx.Beckhoff_ER7xxx.Beckhoff_ER7xxxEK1122.A_0008_ER7041_3002_0022.STM_Velocity.Velocity <-> STM Velocity/Velocity
//     PlcTask Inputs/GVL_iXlinker.EtherCAT_Master_ERxxxx.Beckhoff_ER7xxx.Beckhoff_ER7xxxEK1122.A_0008_ER7041_3002_0022.WcState.WcState <-> WcState/WcState
//     PlcTask Inputs/GVL_iXlinker.EtherCAT_Master_ERxxxx.Beckhoff_ER7xxx.Beckhoff_ER7xxxEK1122.A_0008_ER7041_3002_0022.WcState.InputToggle <-> WcState/InputToggle
//     PlcTask Inputs/GVL_iXlinker.EtherCAT_Master_ERxxxx.Beckhoff_ER7xxx.Beckhoff_ER7xxxEK1122.A_0008_ER7041_3002_0022.InfoData.AdsAddr <-> InfoData/AdsAddr
//     PlcTask Inputs/GVL_iXlinker.EtherCAT_Master_ERxxxx.Beckhoff_ER7xxx.Beckhoff_ER7xxxEK1122.A_0008_ER7041_3002_0022.InfoData.Chn0 <-> InfoData/Chn0
//     PlcTask Inputs/GVL_iXlinker.EtherCAT_Master_ERxxxx.Beckhoff_ER7xxx.Beckhoff_ER7xxxEK1122.A_0008_ER7041_3002_0022.InfoData.Chn1 <-> InfoData/Chn1
//     PlcTask Inputs/GVL_iXlinker.EtherCAT_Master_ERxxxx.Beckhoff_ER7xxx.Beckhoff_ER7xxxEK1122.A_0008_ER7041_3002_0022.InfoData.State <-> InfoData/State
//   PLC/PLC Instance <-> EtherCAT Master ERxxxx/Beckhoff ER7xxx/Beckhoff ER7xxxEK1122/A_0009(ER7342-0002-0020)
//     PlcTask Inputs/GVL_iXlinker.EtherCAT_Master_ERxxxx.Beckhoff_ER7xxx.Beckhoff_ER7xxxEK1122.A_0009_ER7342_0002_0020.ENC_Status_compact_Channel_1.Status/Latch_extern_valid <-> ENC Status compact Channel 1/Status/Latch extern valid
//     PlcTask Inputs/GVL_iXlinker.EtherCAT_Master_ERxxxx.Beckhoff_ER7xxx.Beckhoff_ER7xxxEK1122.A_0009_ER7342_0002_0020.ENC_Status_compact_Channel_2.Status/Latch_extern_valid <-> ENC Status compact Channel 2/Status/Latch extern valid
//     PlcTask Inputs/GVL_iXlinker.EtherCAT_Master_ERxxxx.Beckhoff_ER7xxx.Beckhoff_ER7xxxEK1122.A_0009_ER7342_0002_0020.ENC_Status_compact_Channel_1.Status/Set_counter_done <-> ENC Status compact Channel 1/Status/Set counter done
//     PlcTask Inputs/GVL_iXlinker.EtherCAT_Master_ERxxxx.Beckhoff_ER7xxx.Beckhoff_ER7xxxEK1122.A_0009_ER7342_0002_0020.ENC_Status_compact_Channel_2.Status/Set_counter_done <-> ENC Status compact Channel 2/Status/Set counter done
//     PlcTask Inputs/GVL_iXlinker.EtherCAT_Master_ERxxxx.Beckhoff_ER7xxx.Beckhoff_ER7xxxEK1122.A_0009_ER7342_0002_0020.ENC_Status_compact_Channel_1.Status/Counter_underflow <-> ENC Status compact Channel 1/Status/Counter underflow
//     PlcTask Inputs/GVL_iXlinker.EtherCAT_Master_ERxxxx.Beckhoff_ER7xxx.Beckhoff_ER7xxxEK1122.A_0009_ER7342_0002_0020.ENC_Status_compact_Channel_2.Status/Counter_underflow <-> ENC Status compact Channel 2/Status/Counter underflow
//     PlcTask Inputs/GVL_iXlinker.EtherCAT_Master_ERxxxx.Beckhoff_ER7xxx.Beckhoff_ER7xxxEK1122.A_0009_ER7342_0002_0020.ENC_Status_compact_Channel_1.Status/Counter_overflow <-> ENC Status compact Channel 1/Status/Counter overflow
//     PlcTask Inputs/GVL_iXlinker.EtherCAT_Master_ERxxxx.Beckhoff_ER7xxx.Beckhoff_ER7xxxEK1122.A_0009_ER7342_0002_0020.ENC_Status_compact_Channel_2.Status/Counter_overflow <-> ENC Status compact Channel 2/Status/Counter overflow
//     PlcTask Inputs/GVL_iXlinker.EtherCAT_Master_ERxxxx.Beckhoff_ER7xxx.Beckhoff_ER7xxxEK1122.A_0009_ER7342_0002_0020.ENC_Status_compact_Channel_1.Status/Extrapolation_stall <-> ENC Status compact Channel 1/Status/Extrapolation stall
//     PlcTask Inputs/GVL_iXlinker.EtherCAT_Master_ERxxxx.Beckhoff_ER7xxx.Beckhoff_ER7xxxEK1122.A_0009_ER7342_0002_0020.ENC_Status_compact_Channel_2.Status/Extrapolation_stall <-> ENC Status compact Channel 2/Status/Extrapolation stall
//     PlcTask Inputs/GVL_iXlinker.EtherCAT_Master_ERxxxx.Beckhoff_ER7xxx.Beckhoff_ER7xxxEK1122.A_0009_ER7342_0002_0020.ENC_Status_compact_Channel_1.Status/Status_of_input_A <-> ENC Status compact Channel 1/Status/Status of input A
//     PlcTask Inputs/GVL_iXlinker.EtherCAT_Master_ERxxxx.Beckhoff_ER7xxx.Beckhoff_ER7xxxEK1122.A_0009_ER7342_0002_0020.ENC_Status_compact_Channel_2.Status/Status_of_input_A <-> ENC Status compact Channel 2/Status/Status of input A
//     PlcTask Inputs/GVL_iXlinker.EtherCAT_Master_ERxxxx.Beckhoff_ER7xxx.Beckhoff_ER7xxxEK1122.A_0009_ER7342_0002_0020.ENC_Status_compact_Channel_1.Status/Status_of_input_B <-> ENC Status compact Channel 1/Status/Status of input B
//     PlcTask Inputs/GVL_iXlinker.EtherCAT_Master_ERxxxx.Beckhoff_ER7xxx.Beckhoff_ER7xxxEK1122.A_0009_ER7342_0002_0020.ENC_Status_compact_Channel_2.Status/Status_of_input_B <-> ENC Status compact Channel 2/Status/Status of input B
//     PlcTask Inputs/GVL_iXlinker.EtherCAT_Master_ERxxxx.Beckhoff_ER7xxx.Beckhoff_ER7xxxEK1122.A_0009_ER7342_0002_0020.ENC_Status_compact_Channel_1.Status/Status_of_extern_latch <-> ENC Status compact Channel 1/Status/Status of extern latch
//     PlcTask Inputs/GVL_iXlinker.EtherCAT_Master_ERxxxx.Beckhoff_ER7xxx.Beckhoff_ER7xxxEK1122.A_0009_ER7342_0002_0020.ENC_Status_compact_Channel_2.Status/Status_of_extern_latch <-> ENC Status compact Channel 2/Status/Status of extern latch
//     PlcTask Inputs/GVL_iXlinker.EtherCAT_Master_ERxxxx.Beckhoff_ER7xxx.Beckhoff_ER7xxxEK1122.A_0009_ER7342_0002_0020.ENC_Status_compact_Channel_1.Status/Sync_error <-> ENC Status compact Channel 1/Status/Sync error
//     PlcTask Inputs/GVL_iXlinker.EtherCAT_Master_ERxxxx.Beckhoff_ER7xxx.Beckhoff_ER7xxxEK1122.A_0009_ER7342_0002_0020.ENC_Status_compact_Channel_2.Status/Sync_error <-> ENC Status compact Channel 2/Status/Sync error
//     PlcTask Inputs/GVL_iXlinker.EtherCAT_Master_ERxxxx.Beckhoff_ER7xxx.Beckhoff_ER7xxxEK1122.A_0009_ER7342_0002_0020.ENC_Status_compact_Channel_1.Status/TxPDO_Toggle <-> ENC Status compact Channel 1/Status/TxPDO Toggle
//     PlcTask Inputs/GVL_iXlinker.EtherCAT_Master_ERxxxx.Beckhoff_ER7xxx.Beckhoff_ER7xxxEK1122.A_0009_ER7342_0002_0020.ENC_Status_compact_Channel_2.Status/TxPDO_Toggle <-> ENC Status compact Channel 2/Status/TxPDO Toggle
//     PlcTask Inputs/GVL_iXlinker.EtherCAT_Master_ERxxxx.Beckhoff_ER7xxx.Beckhoff_ER7xxxEK1122.A_0009_ER7342_0002_0020.ENC_Status_compact_Channel_1.Counter_value <-> ENC Status compact Channel 1/Counter value
//     PlcTask Inputs/GVL_iXlinker.EtherCAT_Master_ERxxxx.Beckhoff_ER7xxx.Beckhoff_ER7xxxEK1122.A_0009_ER7342_0002_0020.ENC_Status_compact_Channel_2.Counter_value <-> ENC Status compact Channel 2/Counter value
//     PlcTask Inputs/GVL_iXlinker.EtherCAT_Master_ERxxxx.Beckhoff_ER7xxx.Beckhoff_ER7xxxEK1122.A_0009_ER7342_0002_0020.ENC_Status_compact_Channel_1.Latch_value <-> ENC Status compact Channel 1/Latch value
//     PlcTask Inputs/GVL_iXlinker.EtherCAT_Master_ERxxxx.Beckhoff_ER7xxx.Beckhoff_ER7xxxEK1122.A_0009_ER7342_0002_0020.ENC_Status_compact_Channel_2.Latch_value <-> ENC Status compact Channel 2/Latch value
//     PlcTask Inputs/GVL_iXlinker.EtherCAT_Master_ERxxxx.Beckhoff_ER7xxx.Beckhoff_ER7xxxEK1122.A_0009_ER7342_0002_0020.DCM_Status_Channel_1.Status/Ready_to_enable <-> DCM Status Channel 1/Status/Ready to enable
//     PlcTask Inputs/GVL_iXlinker.EtherCAT_Master_ERxxxx.Beckhoff_ER7xxx.Beckhoff_ER7xxxEK1122.A_0009_ER7342_0002_0020.DCM_Status_Channel_2.Status/Ready_to_enable <-> DCM Status Channel 2/Status/Ready to enable
//     PlcTask Inputs/GVL_iXlinker.EtherCAT_Master_ERxxxx.Beckhoff_ER7xxx.Beckhoff_ER7xxxEK1122.A_0009_ER7342_0002_0020.DCM_Status_Channel_1.Status/Ready <-> DCM Status Channel 1/Status/Ready
//     PlcTask Inputs/GVL_iXlinker.EtherCAT_Master_ERxxxx.Beckhoff_ER7xxx.Beckhoff_ER7xxxEK1122.A_0009_ER7342_0002_0020.DCM_Status_Channel_2.Status/Ready <-> DCM Status Channel 2/Status/Ready
//     PlcTask Inputs/GVL_iXlinker.EtherCAT_Master_ERxxxx.Beckhoff_ER7xxx.Beckhoff_ER7xxxEK1122.A_0009_ER7342_0002_0020.DCM_Status_Channel_1.Status/Warning <-> DCM Status Channel 1/Status/Warning
//     PlcTask Inputs/GVL_iXlinker.EtherCAT_Master_ERxxxx.Beckhoff_ER7xxx.Beckhoff_ER7xxxEK1122.A_0009_ER7342_0002_0020.DCM_Status_Channel_2.Status/Warning <-> DCM Status Channel 2/Status/Warning
//     PlcTask Inputs/GVL_iXlinker.EtherCAT_Master_ERxxxx.Beckhoff_ER7xxx.Beckhoff_ER7xxxEK1122.A_0009_ER7342_0002_0020.DCM_Status_Channel_1.Status/Error <-> DCM Status Channel 1/Status/Error
//     PlcTask Inputs/GVL_iXlinker.EtherCAT_Master_ERxxxx.Beckhoff_ER7xxx.Beckhoff_ER7xxxEK1122.A_0009_ER7342_0002_0020.DCM_Status_Channel_2.Status/Error <-> DCM Status Channel 2/Status/Error
//     PlcTask Inputs/GVL_iXlinker.EtherCAT_Master_ERxxxx.Beckhoff_ER7xxx.Beckhoff_ER7xxxEK1122.A_0009_ER7342_0002_0020.DCM_Status_Channel_1.Status/Moving_positive <-> DCM Status Channel 1/Status/Moving positive
//     PlcTask Inputs/GVL_iXlinker.EtherCAT_Master_ERxxxx.Beckhoff_ER7xxx.Beckhoff_ER7xxxEK1122.A_0009_ER7342_0002_0020.DCM_Status_Channel_2.Status/Moving_positive <-> DCM Status Channel 2/Status/Moving positive
//     PlcTask Inputs/GVL_iXlinker.EtherCAT_Master_ERxxxx.Beckhoff_ER7xxx.Beckhoff_ER7xxxEK1122.A_0009_ER7342_0002_0020.DCM_Status_Channel_1.Status/Moving_negative <-> DCM Status Channel 1/Status/Moving negative
//     PlcTask Inputs/GVL_iXlinker.EtherCAT_Master_ERxxxx.Beckhoff_ER7xxx.Beckhoff_ER7xxxEK1122.A_0009_ER7342_0002_0020.DCM_Status_Channel_2.Status/Moving_negative <-> DCM Status Channel 2/Status/Moving negative
//     PlcTask Inputs/GVL_iXlinker.EtherCAT_Master_ERxxxx.Beckhoff_ER7xxx.Beckhoff_ER7xxxEK1122.A_0009_ER7342_0002_0020.DCM_Status_Channel_1.Status/Torque_reduced <-> DCM Status Channel 1/Status/Torque reduced
//     PlcTask Inputs/GVL_iXlinker.EtherCAT_Master_ERxxxx.Beckhoff_ER7xxx.Beckhoff_ER7xxxEK1122.A_0009_ER7342_0002_0020.DCM_Status_Channel_2.Status/Torque_reduced <-> DCM Status Channel 2/Status/Torque reduced
//     PlcTask Inputs/GVL_iXlinker.EtherCAT_Master_ERxxxx.Beckhoff_ER7xxx.Beckhoff_ER7xxxEK1122.A_0009_ER7342_0002_0020.DCM_Status_Channel_1.Status/Digital_input_1 <-> DCM Status Channel 1/Status/Digital input 1
//     PlcTask Inputs/GVL_iXlinker.EtherCAT_Master_ERxxxx.Beckhoff_ER7xxx.Beckhoff_ER7xxxEK1122.A_0009_ER7342_0002_0020.DCM_Status_Channel_1.Status/Digital_input_2 <-> DCM Status Channel 1/Status/Digital input 2
//     PlcTask Inputs/GVL_iXlinker.EtherCAT_Master_ERxxxx.Beckhoff_ER7xxx.Beckhoff_ER7xxxEK1122.A_0009_ER7342_0002_0020.DCM_Status_Channel_2.Status/Digital_input_1 <-> DCM Status Channel 2/Status/Digital input 1
//     PlcTask Inputs/GVL_iXlinker.EtherCAT_Master_ERxxxx.Beckhoff_ER7xxx.Beckhoff_ER7xxxEK1122.A_0009_ER7342_0002_0020.DCM_Status_Channel_2.Status/Digital_input_2 <-> DCM Status Channel 2/Status/Digital input 2
//     PlcTask Inputs/GVL_iXlinker.EtherCAT_Master_ERxxxx.Beckhoff_ER7xxx.Beckhoff_ER7xxxEK1122.A_0009_ER7342_0002_0020.DCM_Status_Channel_1.Status/Sync_error <-> DCM Status Channel 1/Status/Sync error
//     PlcTask Inputs/GVL_iXlinker.EtherCAT_Master_ERxxxx.Beckhoff_ER7xxx.Beckhoff_ER7xxxEK1122.A_0009_ER7342_0002_0020.DCM_Status_Channel_2.Status/Sync_error <-> DCM Status Channel 2/Status/Sync error
//     PlcTask Inputs/GVL_iXlinker.EtherCAT_Master_ERxxxx.Beckhoff_ER7xxx.Beckhoff_ER7xxxEK1122.A_0009_ER7342_0002_0020.DCM_Status_Channel_1.Status/TxPDO_Toggle <-> DCM Status Channel 1/Status/TxPDO Toggle
//     PlcTask Inputs/GVL_iXlinker.EtherCAT_Master_ERxxxx.Beckhoff_ER7xxx.Beckhoff_ER7xxxEK1122.A_0009_ER7342_0002_0020.DCM_Status_Channel_2.Status/TxPDO_Toggle <-> DCM Status Channel 2/Status/TxPDO Toggle
//     PlcTask Outputs/GVL_iXlinker.EtherCAT_Master_ERxxxx.Beckhoff_ER7xxx.Beckhoff_ER7xxxEK1122.A_0009_ER7342_0002_0020.ENC_Control_compact_Channel_1.Control/Enable_latch_extern_on_positive_edge <-> ENC Control compact Channel 1/Control/Enable latch extern on positive edge
//     PlcTask Outputs/GVL_iXlinker.EtherCAT_Master_ERxxxx.Beckhoff_ER7xxx.Beckhoff_ER7xxxEK1122.A_0009_ER7342_0002_0020.ENC_Control_compact_Channel_2.Control/Enable_latch_extern_on_positive_edge <-> ENC Control compact Channel 2/Control/Enable latch extern on positive edge
//     PlcTask Outputs/GVL_iXlinker.EtherCAT_Master_ERxxxx.Beckhoff_ER7xxx.Beckhoff_ER7xxxEK1122.A_0009_ER7342_0002_0020.ENC_Control_compact_Channel_1.Control/Set_counter <-> ENC Control compact Channel 1/Control/Set counter
//     PlcTask Outputs/GVL_iXlinker.EtherCAT_Master_ERxxxx.Beckhoff_ER7xxx.Beckhoff_ER7xxxEK1122.A_0009_ER7342_0002_0020.ENC_Control_compact_Channel_2.Control/Set_counter <-> ENC Control compact Channel 2/Control/Set counter
//     PlcTask Outputs/GVL_iXlinker.EtherCAT_Master_ERxxxx.Beckhoff_ER7xxx.Beckhoff_ER7xxxEK1122.A_0009_ER7342_0002_0020.ENC_Control_compact_Channel_1.Control/Enable_latch_extern_on_negative_edge <-> ENC Control compact Channel 1/Control/Enable latch extern on negative edge
//     PlcTask Outputs/GVL_iXlinker.EtherCAT_Master_ERxxxx.Beckhoff_ER7xxx.Beckhoff_ER7xxxEK1122.A_0009_ER7342_0002_0020.ENC_Control_compact_Channel_2.Control/Enable_latch_extern_on_negative_edge <-> ENC Control compact Channel 2/Control/Enable latch extern on negative edge
//     PlcTask Outputs/GVL_iXlinker.EtherCAT_Master_ERxxxx.Beckhoff_ER7xxx.Beckhoff_ER7xxxEK1122.A_0009_ER7342_0002_0020.ENC_Control_compact_Channel_1.Set_counter_value <-> ENC Control compact Channel 1/Set counter value
//     PlcTask Outputs/GVL_iXlinker.EtherCAT_Master_ERxxxx.Beckhoff_ER7xxx.Beckhoff_ER7xxxEK1122.A_0009_ER7342_0002_0020.ENC_Control_compact_Channel_2.Set_counter_value <-> ENC Control compact Channel 2/Set counter value
//     PlcTask Outputs/GVL_iXlinker.EtherCAT_Master_ERxxxx.Beckhoff_ER7xxx.Beckhoff_ER7xxxEK1122.A_0009_ER7342_0002_0020.DCM_Control_Channel_1.Control/Enable <-> DCM Control Channel 1/Control/Enable
//     PlcTask Outputs/GVL_iXlinker.EtherCAT_Master_ERxxxx.Beckhoff_ER7xxx.Beckhoff_ER7xxxEK1122.A_0009_ER7342_0002_0020.DCM_Control_Channel_2.Control/Enable <-> DCM Control Channel 2/Control/Enable
//     PlcTask Outputs/GVL_iXlinker.EtherCAT_Master_ERxxxx.Beckhoff_ER7xxx.Beckhoff_ER7xxxEK1122.A_0009_ER7342_0002_0020.DCM_Control_Channel_1.Control/Reset <-> DCM Control Channel 1/Control/Reset
//     PlcTask Outputs/GVL_iXlinker.EtherCAT_Master_ERxxxx.Beckhoff_ER7xxx.Beckhoff_ER7xxxEK1122.A_0009_ER7342_0002_0020.DCM_Control_Channel_2.Control/Reset <-> DCM Control Channel 2/Control/Reset
//     PlcTask Outputs/GVL_iXlinker.EtherCAT_Master_ERxxxx.Beckhoff_ER7xxx.Beckhoff_ER7xxxEK1122.A_0009_ER7342_0002_0020.DCM_Control_Channel_1.Control/Reduce_torque <-> DCM Control Channel 1/Control/Reduce torque
//     PlcTask Outputs/GVL_iXlinker.EtherCAT_Master_ERxxxx.Beckhoff_ER7xxx.Beckhoff_ER7xxxEK1122.A_0009_ER7342_0002_0020.DCM_Control_Channel_2.Control/Reduce_torque <-> DCM Control Channel 2/Control/Reduce torque
//     PlcTask Outputs/GVL_iXlinker.EtherCAT_Master_ERxxxx.Beckhoff_ER7xxx.Beckhoff_ER7xxxEK1122.A_0009_ER7342_0002_0020.DCM_Velocity_Channel_1.Velocity <-> DCM Velocity Channel 1/Velocity
//     PlcTask Outputs/GVL_iXlinker.EtherCAT_Master_ERxxxx.Beckhoff_ER7xxx.Beckhoff_ER7xxxEK1122.A_0009_ER7342_0002_0020.DCM_Velocity_Channel_2.Velocity <-> DCM Velocity Channel 2/Velocity
//     PlcTask Inputs/GVL_iXlinker.EtherCAT_Master_ERxxxx.Beckhoff_ER7xxx.Beckhoff_ER7xxxEK1122.A_0009_ER7342_0002_0020.WcState.WcState <-> WcState/WcState
//     PlcTask Inputs/GVL_iXlinker.EtherCAT_Master_ERxxxx.Beckhoff_ER7xxx.Beckhoff_ER7xxxEK1122.A_0009_ER7342_0002_0020.WcState.InputToggle <-> WcState/InputToggle
//     PlcTask Inputs/GVL_iXlinker.EtherCAT_Master_ERxxxx.Beckhoff_ER7xxx.Beckhoff_ER7xxxEK1122.A_0009_ER7342_0002_0020.InfoData.AdsAddr <-> InfoData/AdsAddr
//     PlcTask Inputs/GVL_iXlinker.EtherCAT_Master_ERxxxx.Beckhoff_ER7xxx.Beckhoff_ER7xxxEK1122.A_0009_ER7342_0002_0020.InfoData.Chn0 <-> InfoData/Chn0
//     PlcTask Inputs/GVL_iXlinker.EtherCAT_Master_ERxxxx.Beckhoff_ER7xxx.Beckhoff_ER7xxxEK1122.A_0009_ER7342_0002_0020.InfoData.Chn1 <-> InfoData/Chn1
//     PlcTask Inputs/GVL_iXlinker.EtherCAT_Master_ERxxxx.Beckhoff_ER7xxx.Beckhoff_ER7xxxEK1122.A_0009_ER7342_0002_0020.InfoData.Chn2 <-> InfoData/Chn2
//     PlcTask Inputs/GVL_iXlinker.EtherCAT_Master_ERxxxx.Beckhoff_ER7xxx.Beckhoff_ER7xxxEK1122.A_0009_ER7342_0002_0020.InfoData.Chn3 <-> InfoData/Chn3
//     PlcTask Inputs/GVL_iXlinker.EtherCAT_Master_ERxxxx.Beckhoff_ER7xxx.Beckhoff_ER7xxxEK1122.A_0009_ER7342_0002_0020.InfoData.State <-> InfoData/State
//   PLC/PLC Instance <-> EtherCAT Master ERxxxx/Beckhoff ER7xxx/Beckhoff ER7xxxEK1122/A_0010(ER7342-0002-0021)
//     PlcTask Inputs/GVL_iXlinker.EtherCAT_Master_ERxxxx.Beckhoff_ER7xxx.Beckhoff_ER7xxxEK1122.A_0010_ER7342_0002_0021.ENC_Status_compact_Channel_1.Status/Latch_extern_valid <-> ENC Status compact Channel 1/Status/Latch extern valid
//     PlcTask Inputs/GVL_iXlinker.EtherCAT_Master_ERxxxx.Beckhoff_ER7xxx.Beckhoff_ER7xxxEK1122.A_0010_ER7342_0002_0021.ENC_Status_compact_Channel_2.Status/Latch_extern_valid <-> ENC Status compact Channel 2/Status/Latch extern valid
//     PlcTask Inputs/GVL_iXlinker.EtherCAT_Master_ERxxxx.Beckhoff_ER7xxx.Beckhoff_ER7xxxEK1122.A_0010_ER7342_0002_0021.ENC_Status_compact_Channel_1.Status/Set_counter_done <-> ENC Status compact Channel 1/Status/Set counter done
//     PlcTask Inputs/GVL_iXlinker.EtherCAT_Master_ERxxxx.Beckhoff_ER7xxx.Beckhoff_ER7xxxEK1122.A_0010_ER7342_0002_0021.ENC_Status_compact_Channel_2.Status/Set_counter_done <-> ENC Status compact Channel 2/Status/Set counter done
//     PlcTask Inputs/GVL_iXlinker.EtherCAT_Master_ERxxxx.Beckhoff_ER7xxx.Beckhoff_ER7xxxEK1122.A_0010_ER7342_0002_0021.ENC_Status_compact_Channel_1.Status/Counter_underflow <-> ENC Status compact Channel 1/Status/Counter underflow
//     PlcTask Inputs/GVL_iXlinker.EtherCAT_Master_ERxxxx.Beckhoff_ER7xxx.Beckhoff_ER7xxxEK1122.A_0010_ER7342_0002_0021.ENC_Status_compact_Channel_2.Status/Counter_underflow <-> ENC Status compact Channel 2/Status/Counter underflow
//     PlcTask Inputs/GVL_iXlinker.EtherCAT_Master_ERxxxx.Beckhoff_ER7xxx.Beckhoff_ER7xxxEK1122.A_0010_ER7342_0002_0021.ENC_Status_compact_Channel_1.Status/Counter_overflow <-> ENC Status compact Channel 1/Status/Counter overflow
//     PlcTask Inputs/GVL_iXlinker.EtherCAT_Master_ERxxxx.Beckhoff_ER7xxx.Beckhoff_ER7xxxEK1122.A_0010_ER7342_0002_0021.ENC_Status_compact_Channel_2.Status/Counter_overflow <-> ENC Status compact Channel 2/Status/Counter overflow
//     PlcTask Inputs/GVL_iXlinker.EtherCAT_Master_ERxxxx.Beckhoff_ER7xxx.Beckhoff_ER7xxxEK1122.A_0010_ER7342_0002_0021.ENC_Status_compact_Channel_1.Status/Extrapolation_stall <-> ENC Status compact Channel 1/Status/Extrapolation stall
//     PlcTask Inputs/GVL_iXlinker.EtherCAT_Master_ERxxxx.Beckhoff_ER7xxx.Beckhoff_ER7xxxEK1122.A_0010_ER7342_0002_0021.ENC_Status_compact_Channel_2.Status/Extrapolation_stall <-> ENC Status compact Channel 2/Status/Extrapolation stall
//     PlcTask Inputs/GVL_iXlinker.EtherCAT_Master_ERxxxx.Beckhoff_ER7xxx.Beckhoff_ER7xxxEK1122.A_0010_ER7342_0002_0021.ENC_Status_compact_Channel_1.Status/Status_of_input_A <-> ENC Status compact Channel 1/Status/Status of input A
//     PlcTask Inputs/GVL_iXlinker.EtherCAT_Master_ERxxxx.Beckhoff_ER7xxx.Beckhoff_ER7xxxEK1122.A_0010_ER7342_0002_0021.ENC_Status_compact_Channel_2.Status/Status_of_input_A <-> ENC Status compact Channel 2/Status/Status of input A
//     PlcTask Inputs/GVL_iXlinker.EtherCAT_Master_ERxxxx.Beckhoff_ER7xxx.Beckhoff_ER7xxxEK1122.A_0010_ER7342_0002_0021.ENC_Status_compact_Channel_1.Status/Status_of_input_B <-> ENC Status compact Channel 1/Status/Status of input B
//     PlcTask Inputs/GVL_iXlinker.EtherCAT_Master_ERxxxx.Beckhoff_ER7xxx.Beckhoff_ER7xxxEK1122.A_0010_ER7342_0002_0021.ENC_Status_compact_Channel_2.Status/Status_of_input_B <-> ENC Status compact Channel 2/Status/Status of input B
//     PlcTask Inputs/GVL_iXlinker.EtherCAT_Master_ERxxxx.Beckhoff_ER7xxx.Beckhoff_ER7xxxEK1122.A_0010_ER7342_0002_0021.ENC_Status_compact_Channel_1.Status/Status_of_extern_latch <-> ENC Status compact Channel 1/Status/Status of extern latch
//     PlcTask Inputs/GVL_iXlinker.EtherCAT_Master_ERxxxx.Beckhoff_ER7xxx.Beckhoff_ER7xxxEK1122.A_0010_ER7342_0002_0021.ENC_Status_compact_Channel_2.Status/Status_of_extern_latch <-> ENC Status compact Channel 2/Status/Status of extern latch
//     PlcTask Inputs/GVL_iXlinker.EtherCAT_Master_ERxxxx.Beckhoff_ER7xxx.Beckhoff_ER7xxxEK1122.A_0010_ER7342_0002_0021.ENC_Status_compact_Channel_1.Status/Sync_error <-> ENC Status compact Channel 1/Status/Sync error
//     PlcTask Inputs/GVL_iXlinker.EtherCAT_Master_ERxxxx.Beckhoff_ER7xxx.Beckhoff_ER7xxxEK1122.A_0010_ER7342_0002_0021.ENC_Status_compact_Channel_2.Status/Sync_error <-> ENC Status compact Channel 2/Status/Sync error
//     PlcTask Inputs/GVL_iXlinker.EtherCAT_Master_ERxxxx.Beckhoff_ER7xxx.Beckhoff_ER7xxxEK1122.A_0010_ER7342_0002_0021.ENC_Status_compact_Channel_1.Status/TxPDO_Toggle <-> ENC Status compact Channel 1/Status/TxPDO Toggle
//     PlcTask Inputs/GVL_iXlinker.EtherCAT_Master_ERxxxx.Beckhoff_ER7xxx.Beckhoff_ER7xxxEK1122.A_0010_ER7342_0002_0021.ENC_Status_compact_Channel_2.Status/TxPDO_Toggle <-> ENC Status compact Channel 2/Status/TxPDO Toggle
//     PlcTask Inputs/GVL_iXlinker.EtherCAT_Master_ERxxxx.Beckhoff_ER7xxx.Beckhoff_ER7xxxEK1122.A_0010_ER7342_0002_0021.ENC_Status_compact_Channel_1.Counter_value <-> ENC Status compact Channel 1/Counter value
//     PlcTask Inputs/GVL_iXlinker.EtherCAT_Master_ERxxxx.Beckhoff_ER7xxx.Beckhoff_ER7xxxEK1122.A_0010_ER7342_0002_0021.ENC_Status_compact_Channel_2.Counter_value <-> ENC Status compact Channel 2/Counter value
//     PlcTask Inputs/GVL_iXlinker.EtherCAT_Master_ERxxxx.Beckhoff_ER7xxx.Beckhoff_ER7xxxEK1122.A_0010_ER7342_0002_0021.ENC_Status_compact_Channel_1.Latch_value <-> ENC Status compact Channel 1/Latch value
//     PlcTask Inputs/GVL_iXlinker.EtherCAT_Master_ERxxxx.Beckhoff_ER7xxx.Beckhoff_ER7xxxEK1122.A_0010_ER7342_0002_0021.ENC_Status_compact_Channel_2.Latch_value <-> ENC Status compact Channel 2/Latch value
//     PlcTask Inputs/GVL_iXlinker.EtherCAT_Master_ERxxxx.Beckhoff_ER7xxx.Beckhoff_ER7xxxEK1122.A_0010_ER7342_0002_0021.DCM_Status_Channel_1.Status/Ready_to_enable <-> DCM Status Channel 1/Status/Ready to enable
//     PlcTask Inputs/GVL_iXlinker.EtherCAT_Master_ERxxxx.Beckhoff_ER7xxx.Beckhoff_ER7xxxEK1122.A_0010_ER7342_0002_0021.DCM_Status_Channel_2.Status/Ready_to_enable <-> DCM Status Channel 2/Status/Ready to enable
//     PlcTask Inputs/GVL_iXlinker.EtherCAT_Master_ERxxxx.Beckhoff_ER7xxx.Beckhoff_ER7xxxEK1122.A_0010_ER7342_0002_0021.DCM_Status_Channel_1.Status/Ready <-> DCM Status Channel 1/Status/Ready
//     PlcTask Inputs/GVL_iXlinker.EtherCAT_Master_ERxxxx.Beckhoff_ER7xxx.Beckhoff_ER7xxxEK1122.A_0010_ER7342_0002_0021.DCM_Status_Channel_2.Status/Ready <-> DCM Status Channel 2/Status/Ready
//     PlcTask Inputs/GVL_iXlinker.EtherCAT_Master_ERxxxx.Beckhoff_ER7xxx.Beckhoff_ER7xxxEK1122.A_0010_ER7342_0002_0021.DCM_Status_Channel_1.Status/Warning <-> DCM Status Channel 1/Status/Warning
//     PlcTask Inputs/GVL_iXlinker.EtherCAT_Master_ERxxxx.Beckhoff_ER7xxx.Beckhoff_ER7xxxEK1122.A_0010_ER7342_0002_0021.DCM_Status_Channel_2.Status/Warning <-> DCM Status Channel 2/Status/Warning
//     PlcTask Inputs/GVL_iXlinker.EtherCAT_Master_ERxxxx.Beckhoff_ER7xxx.Beckhoff_ER7xxxEK1122.A_0010_ER7342_0002_0021.DCM_Status_Channel_1.Status/Error <-> DCM Status Channel 1/Status/Error
//     PlcTask Inputs/GVL_iXlinker.EtherCAT_Master_ERxxxx.Beckhoff_ER7xxx.Beckhoff_ER7xxxEK1122.A_0010_ER7342_0002_0021.DCM_Status_Channel_2.Status/Error <-> DCM Status Channel 2/Status/Error
